LIN {X 0,Y 383.71,Z 437.211,A -85,B 0,C 180,E1 -14302.123,E2 -14302.123} C_VEL
LIN {X 0,Y 386.289,Z 439.249,A -85,B 0,C 180,E1 -14303.895,E2 -14303.895} C_VEL
LIN {X 0,Y 388.386,Z 440.41,A -85,B 0,C 180,E1 -14305.849,E2 -14305.849} C_VEL
LIN {X 0,Y 389.529,Z 440.796,A -85,B 0,C 180,E1 -14307.433,E2 -14307.433} C_VEL
LIN {X 0,Y 390.099,Z 441.222,A -85,B 0,C 180,E1 -14308.967,E2 -14308.967} C_VEL
LIN {X 0,Y 390.27,Z 441.152,A -85,B 0,C 180,E1 -14310,E2 -14310} C_VEL
LIN {X 0,Y 389.995,Z 441.089,A -85,B 0,C 180,E1 -14311.549,E2 -14311.549} C_VEL
LIN {X 0,Y 389.238,Z 440.657,A -85,B 0,C 180,E1 -14313.105,E2 -14313.105} C_VEL
LIN {X 0,Y 387.614,Z 440.065,A -85,B 0,C 180,E1 -14314.94,E2 -14314.94} C_VEL
LIN {X 0,Y 385.471,Z 438.704,A -85,B 0,C 180,E1 -14316.685,E2 -14316.685} C_VEL
LIN {X 0,Y 383.224,Z 436.724,A -85,B 0,C 180,E1 -14318.162,E2 -14318.162} C_VEL
LIN {X 0,Y 380.545,Z 433.68,A -85,B 0,C 180,E1 -14319.669,E2 -14319.669} C_VEL
LIN {X 0,Y 377.343,Z 431.776,A -85,B 0,C 180,E1 -14321.118,E2 -14321.118} C_VEL
LIN {X 0,Y 373.996,Z 428.62,A -85,B 0,C 180,E1 -14322.503,E2 -14322.503} C_VEL
LIN {X 0,Y 371.832,Z 426.329,A -85,B 0,C 180,E1 -14323.336,E2 -14323.336} C_VEL
LIN {X 0,Y 368.143,Z 423.337,A -85,B 0,C 180,E1 -14324.583,E2 -14324.583} C_VEL
LIN {X 0,Y 365.094,Z 419.876,A -85,B 0,C 180,E1 -14325.58,E2 -14325.58} C_VEL
LIN {X 0,Y 361.446,Z 416.759,A -85,B 0,C 180,E1 -14326.666,E2 -14326.666} C_VEL
LIN {X 0,Y 358.551,Z 413.451,A -85,B 0,C 180,E1 -14327.482,E2 -14327.482} C_VEL
LIN {X 0,Y 355.376,Z 410.462,A -85,B 0,C 180,E1 -14328.333,E2 -14328.333} C_VEL
LIN {X 0,Y 353.051,Z 407.518,A -85,B 0,C 180,E1 -14328.94,E2 -14328.94} C_VEL
LIN {X 0,Y 350.002,Z 404.381,A -85,B 0,C 180,E1 -14329.706,E2 -14329.706} C_VEL
LIN {X 0,Y 348.216,Z 401.952,A -85,B 0,C 180,E1 -14330.137,E2 -14330.137} C_VEL
LIN {X 0,Y 345.497,Z 399.057,A -85,B 0,C 180,E1 -14330.784,E2 -14330.784} C_VEL
LIN {X 0,Y 344.016,Z 396.656,A -85,B 0,C 180,E1 -14331.146,E2 -14331.146} C_VEL
LIN {X 0,Y 341.851,Z 394.52,A -85,B 0,C 180,E1 -14331.605,E2 -14331.605} C_VEL
LIN {X 0,Y 340.819,Z 392.08,A -85,B 0,C 180,E1 -14331.984,E2 -14331.984} C_VEL
LIN {X 0,Y 340.741,Z 391.556,A -85,B 0,C 180,E1 -14332.43,E2 -14332.43} C_VEL
LIN {X 0,Y 340.768,Z 391.54,A -85,B 0,C 180,E1 -14335.664,E2 -14335.664} C_VEL
LIN {X 0,Y 340.737,Z 391.527,A -85,B 0,C 180,E1 -14338.319,E2 -14338.319} C_VEL
LIN {X 0,Y 340.698,Z 391.542,A -85,B 0,C 180,E1 -14341.044,E2 -14341.044} C_VEL
LIN {X 0,Y 340.713,Z 391.518,A -85,B 0,C 180,E1 -14345.279,E2 -14345.279} C_VEL
LIN {X 0,Y 340.72,Z 391.546,A -85,B 0,C 180,E1 -14348.389,E2 -14348.389} C_VEL
LIN {X 0,Y 340.699,Z 391.499,A -85,B 0,C 180,E1 -14352.047,E2 -14352.047} C_VEL
LIN {X 0,Y 340.688,Z 391.544,A -85,B 0,C 180,E1 -14355.463,E2 -14355.463} C_VEL
LIN {X 0,Y 340.697,Z 391.534,A -85,B 0,C 180,E1 -14358.693,E2 -14358.693} C_VEL
LIN {X 0,Y 340.734,Z 391.541,A -85,B 0,C 180,E1 -14361.774,E2 -14361.774} C_VEL
LIN {X 0,Y 340.716,Z 391.524,A -85,B 0,C 180,E1 -14365.596,E2 -14365.596} C_VEL
LIN {X 0,Y 340.717,Z 391.542,A -85,B 0,C 180,E1 -14369.566,E2 -14369.566} C_VEL
LIN {X 0,Y 340.799,Z 391.513,A -85,B 0,C 180,E1 -14373.02,E2 -14373.02} C_VEL
LIN {X 0,Y 340.755,Z 391.53,A -85,B 0,C 180,E1 -14374.691,E2 -14374.691} C_VEL
LIN {X 0,Y 340.072,Z 391.623,A -85,B 0,C 180,E1 -14375.678,E2 -14375.678} C_VEL
LIN {X 0,Y 337.177,Z 391.982,A -85,B 0,C 180,E1 -14377.283,E2 -14377.283} C_VEL
LIN {X 0,Y 334.755,Z 392.275,A -85,B 0,C 180,E1 -14378.582,E2 -14378.582} C_VEL
LIN {X 0,Y 333.756,Z 392.392,A -85,B 0,C 180,E1 -14379.589,E2 -14379.589} C_VEL
LIN {X 0,Y 333.695,Z 392.393,A -85,B 0,C 180,E1 -14379.93,E2 -14379.93} C_VEL
LIN {X 0,Y 333.74,Z 392.401,A -85,B 0,C 180,E1 -14382.854,E2 -14382.854} C_VEL
LIN {X 0,Y 333.792,Z 392.401,A -85,B 0,C 180,E1 -14386.609,E2 -14386.609} C_VEL
LIN {X 0,Y 333.858,Z 392.366,A -85,B 0,C 180,E1 -14390.306,E2 -14390.306} C_VEL
LIN {X 0,Y 334.019,Z 392.371,A -85,B 0,C 180,E1 -14392.748,E2 -14392.748} C_VEL
LIN {X 0,Y 333.807,Z 392.402,A -85,B 0,C 180,E1 -14395.17,E2 -14395.17} C_VEL
LIN {X 0,Y 334.102,Z 392.353,A -85,B 0,C 180,E1 -14397.589,E2 -14397.589} C_VEL
LIN {X 0,Y 334.223,Z 392.318,A -85,B 0,C 180,E1 -14400.001,E2 -14400.001} C_VEL
LIN {X 0,Y 334.102,Z 392.358,A -85,B 0,C 180,E1 -14402.412,E2 -14402.412} C_VEL
LIN {X 0,Y 334.022,Z 392.364,A -85,B 0,C 180,E1 -14407.253,E2 -14407.253} C_VEL
LIN {X 0,Y 333.829,Z 392.38,A -85,B 0,C 180,E1 -14410.923,E2 -14410.923} C_VEL
LIN {X 0,Y 333.804,Z 392.401,A -85,B 0,C 180,E1 -14414.635,E2 -14414.635} C_VEL
LIN {X 0,Y 333.792,Z 392.376,A -85,B 0,C 180,E1 -14418.656,E2 -14418.656} C_VEL
LIN {X 0,Y 333.689,Z 392.419,A -85,B 0,C 180,E1 -14422.279,E2 -14422.279} C_VEL
LIN {X 0,Y 333.733,Z 392.389,A -85,B 0,C 180,E1 -14426.247,E2 -14426.247} C_VEL
LIN {X 0,Y 333.709,Z 392.412,A -85,B 0,C 180,E1 -14428.973,E2 -14428.973} C_VEL
LIN {X 0,Y 333.649,Z 392.412,A -85,B 0,C 180,E1 -14432.59,E2 -14432.59} C_VEL
LIN {X 0,Y 333.675,Z 392.417,A -85,B 0,C 180,E1 -14436.14,E2 -14436.14} C_VEL
LIN {X 0,Y 333.683,Z 392.411,A -85,B 0,C 180,E1 -14439.188,E2 -14439.188} C_VEL
LIN {X 0,Y 333.701,Z 392.417,A -85,B 0,C 180,E1 -14442.514,E2 -14442.514} C_VEL
LIN {X 0,Y 333.634,Z 392.428,A -85,B 0,C 180,E1 -14445.962,E2 -14445.962} C_VEL
LIN {X 0,Y 333.646,Z 392.399,A -85,B 0,C 180,E1 -14449.316,E2 -14449.316} C_VEL
LIN {X 0,Y 333.666,Z 392.412,A -85,B 0,C 180,E1 -14453.169,E2 -14453.169} C_VEL
LIN {X 0,Y 333.704,Z 392.564,A -85,B 0,C 180,E1 -14456.865,E2 -14456.865} C_VEL
LIN {X 0,Y 335.043,Z 398.947,A -85,B 0,C 180,E1 -14459.321,E2 -14459.321} C_VEL
LIN {X 0,Y 336.889,Z 408.593,A -85,B 0,C 180,E1 -14462.681,E2 -14462.681} C_VEL
LIN {X 0,Y 337.083,Z 412.536,A -85,B 0,C 180,E1 -14464.035,E2 -14464.035} C_VEL
LIN {X 0,Y 336.305,Z 418.399,A -85,B 0,C 180,E1 -14465.916,E2 -14465.916} C_VEL
LIN {X 0,Y 337.098,Z 422.527,A -85,B 0,C 180,E1 -14466.137,E2 -14466.137} C_VEL
LIN {X 0,Y 341.775,Z 445.874,A -85,B 0,C 180,E1 -14467.003,E2 -14467.003} C_VEL
LIN {X 0,Y 343.729,Z 457.616,A -85,B 0,C 180,E1 -14467.4,E2 -14467.4} C_VEL
LIN {X 0,Y 342.424,Z 523.377,A -85,B 0,C 180,E1 -14468.794,E2 -14468.794} C_VEL
LIN {X 0,Y 341.954,Z 533.264,A -85,B 0,C 180,E1 -14469.118,E2 -14469.118} C_VEL
LIN {X 0,Y 341.257,Z 543.248,A -85,B 0,C 180,E1 -14469.586,E2 -14469.586} C_VEL
LIN {X 0,Y 340.344,Z 553.602,A -85,B 0,C 180,E1 -14470.237,E2 -14470.237} C_VEL
LIN {X 0,Y 339.437,Z 562.747,A -85,B 0,C 180,E1 -14470.968,E2 -14470.968} C_VEL
LIN {X 0,Y 338.37,Z 571.746,A -85,B 0,C 180,E1 -14471.848,E2 -14471.848} C_VEL
LIN {X 0,Y 337.296,Z 580.473,A -85,B 0,C 180,E1 -14472.884,E2 -14472.884} C_VEL
LIN {X 0,Y 336.298,Z 588.415,A -85,B 0,C 180,E1 -14474.013,E2 -14474.013} C_VEL
LIN {X 0,Y 335.243,Z 596.692,A -85,B 0,C 180,E1 -14475.43,E2 -14475.43} C_VEL
LIN {X 0,Y 334.488,Z 602.684,A -85,B 0,C 180,E1 -14476.637,E2 -14476.637} C_VEL
LIN {X 0,Y 333.587,Z 608.993,A -85,B 0,C 180,E1 -14478.147,E2 -14478.147} C_VEL
LIN {X 0,Y 333.006,Z 614.269,A -85,B 0,C 180,E1 -14479.666,E2 -14479.666} C_VEL
LIN {X 0,Y 332.464,Z 619.364,A -85,B 0,C 180,E1 -14481.491,E2 -14481.491} C_VEL
LIN {X 0,Y 332.121,Z 623.328,A -85,B 0,C 180,E1 -14483.317,E2 -14483.317} C_VEL
LIN {X 0,Y 331.981,Z 626.264,A -85,B 0,C 180,E1 -14485.143,E2 -14485.143} C_VEL
LIN {X 0,Y 331.97,Z 627.765,A -85,B 0,C 180,E1 -14486.359,E2 -14486.359} C_VEL
LIN {X 0,Y 331.913,Z 629.287,A -85,B 0,C 180,E1 -14488.787,E2 -14488.787} C_VEL
LIN {X 0,Y 331.953,Z 629.567,A -85,B 0,C 180,E1 -14490,E2 -14490} C_VEL
LIN {X 0,Y 331.916,Z 628.691,A -85,B 0,C 180,E1 -14492.427,E2 -14492.427} C_VEL
LIN {X 0,Y 331.97,Z 627.764,A -85,B 0,C 180,E1 -14493.642,E2 -14493.642} C_VEL
LIN {X 0,Y 332.039,Z 624.416,A -85,B 0,C 180,E1 -14496.075,E2 -14496.075} C_VEL
LIN {X 0,Y 332.335,Z 620.79,A -85,B 0,C 180,E1 -14497.901,E2 -14497.901} C_VEL
LIN {X 0,Y 332.793,Z 616.057,A -85,B 0,C 180,E1 -14499.727,E2 -14499.727} C_VEL
LIN {X 0,Y 333.442,Z 610.083,A -85,B 0,C 180,E1 -14501.551,E2 -14501.551} C_VEL
LIN {X 0,Y 334.289,Z 603.992,A -85,B 0,C 180,E1 -14503.062,E2 -14503.062} C_VEL
LIN {X 0,Y 335.081,Z 598.251,A -85,B 0,C 180,E1 -14504.267,E2 -14504.267} C_VEL
LIN {X 0,Y 336.001,Z 591.595,A -85,B 0,C 180,E1 -14505.467,E2 -14505.467} C_VEL
LIN {X 0,Y 336.919,Z 583.763,A -85,B 0,C 180,E1 -14506.668,E2 -14506.668} C_VEL
LIN {X 0,Y 337.935,Z 575.68,A -85,B 0,C 180,E1 -14507.707,E2 -14507.707} C_VEL
LIN {X 0,Y 339.078,Z 565.919,A -85,B 0,C 180,E1 -14508.74,E2 -14508.74} C_VEL
LIN {X 0,Y 339.985,Z 557.529,A -85,B 0,C 180,E1 -14509.471,E2 -14509.471} C_VEL
LIN {X 0,Y 340.903,Z 547.022,A -85,B 0,C 180,E1 -14510.201,E2 -14510.201} C_VEL
LIN {X 0,Y 341.734,Z 536.691,A -85,B 0,C 180,E1 -14510.739,E2 -14510.739} C_VEL
LIN {X 0,Y 342.353,Z 525.97,A -85,B 0,C 180,E1 -14511.133,E2 -14511.133} C_VEL
LIN {X 0,Y 342.826,Z 503.188,A -85,B 0,C 180,E1 -14511.654,E2 -14511.654} C_VEL
LIN {X 0,Y 343.607,Z 456.424,A -85,B 0,C 180,E1 -14512.635,E2 -14512.635} C_VEL
LIN {X 0,Y 339.119,Z 431.992,A -85,B 0,C 180,E1 -14513.499,E2 -14513.499} C_VEL
LIN {X 0,Y 336.289,Z 418.735,A -85,B 0,C 180,E1 -14514.04,E2 -14514.04} C_VEL
LIN {X 0,Y 336.392,Z 417.243,A -85,B 0,C 180,E1 -14514.403,E2 -14514.403} C_VEL
LIN {X 0,Y 337.206,Z 411.413,A -85,B 0,C 180,E1 -14516.336,E2 -14516.336} C_VEL
LIN {X 0,Y 336.18,Z 404.578,A -85,B 0,C 180,E1 -14518.739,E2 -14518.739} C_VEL
LIN {X 0,Y 334.245,Z 395.104,A -85,B 0,C 180,E1 -14522.173,E2 -14522.173} C_VEL
LIN {X 0,Y 333.705,Z 392.506,A -85,B 0,C 180,E1 -14523.201,E2 -14523.201} C_VEL
LIN {X 0,Y 333.668,Z 392.412,A -85,B 0,C 180,E1 -14526.832,E2 -14526.832} C_VEL
LIN {X 0,Y 333.648,Z 392.398,A -85,B 0,C 180,E1 -14530.767,E2 -14530.767} C_VEL
LIN {X 0,Y 333.645,Z 392.424,A -85,B 0,C 180,E1 -14534.259,E2 -14534.259} C_VEL
LIN {X 0,Y 333.707,Z 392.417,A -85,B 0,C 180,E1 -14537.628,E2 -14537.628} C_VEL
LIN {X 0,Y 333.685,Z 392.412,A -85,B 0,C 180,E1 -14541.195,E2 -14541.195} C_VEL
LIN {X 0,Y 333.687,Z 392.405,A -85,B 0,C 180,E1 -14545.225,E2 -14545.225} C_VEL
LIN {X 0,Y 333.645,Z 392.422,A -85,B 0,C 180,E1 -14548.223,E2 -14548.223} C_VEL
LIN {X 0,Y 333.713,Z 392.411,A -85,B 0,C 180,E1 -14551.027,E2 -14551.027} C_VEL
LIN {X 0,Y 333.736,Z 392.389,A -85,B 0,C 180,E1 -14553.753,E2 -14553.753} C_VEL
LIN {X 0,Y 333.72,Z 392.412,A -85,B 0,C 180,E1 -14557.913,E2 -14557.913} C_VEL
LIN {X 0,Y 333.793,Z 392.376,A -85,B 0,C 180,E1 -14561.589,E2 -14561.589} C_VEL
LIN {X 0,Y 333.808,Z 392.402,A -85,B 0,C 180,E1 -14565.576,E2 -14565.576} C_VEL
LIN {X 0,Y 333.833,Z 392.379,A -85,B 0,C 180,E1 -14569.077,E2 -14569.077} C_VEL
LIN {X 0,Y 334.026,Z 392.364,A -85,B 0,C 180,E1 -14572.747,E2 -14572.747} C_VEL
LIN {X 0,Y 333.81,Z 392.403,A -85,B 0,C 180,E1 -14575.168,E2 -14575.168} C_VEL
LIN {X 0,Y 334.106,Z 392.357,A -85,B 0,C 180,E1 -14577.588,E2 -14577.588} C_VEL
LIN {X 0,Y 334.225,Z 392.317,A -85,B 0,C 180,E1 -14579.999,E2 -14579.999} C_VEL
LIN {X 0,Y 334.106,Z 392.353,A -85,B 0,C 180,E1 -14582.41,E2 -14582.41} C_VEL
LIN {X 0,Y 334.023,Z 392.37,A -85,B 0,C 180,E1 -14587.252,E2 -14587.252} C_VEL
LIN {X 0,Y 333.834,Z 392.372,A -85,B 0,C 180,E1 -14590.921,E2 -14590.921} C_VEL
LIN {X 0,Y 333.806,Z 392.403,A -85,B 0,C 180,E1 -14594.634,E2 -14594.634} C_VEL
LIN {X 0,Y 333.793,Z 392.38,A -85,B 0,C 180,E1 -14598.654,E2 -14598.654} C_VEL
LIN {X 0,Y 333.69,Z 392.416,A -85,B 0,C 180,E1 -14602.278,E2 -14602.278} C_VEL
LIN {X 0,Y 333.732,Z 392.398,A -85,B 0,C 180,E1 -14606.246,E2 -14606.246} C_VEL
LIN {X 0,Y 333.687,Z 392.407,A -85,B 0,C 180,E1 -14608.974,E2 -14608.974} C_VEL
LIN {X 0,Y 333.64,Z 392.422,A -85,B 0,C 180,E1 -14612.586,E2 -14612.586} C_VEL
LIN {X 0,Y 333.674,Z 392.416,A -85,B 0,C 180,E1 -14616.138,E2 -14616.138} C_VEL
LIN {X 0,Y 333.644,Z 392.42,A -85,B 0,C 180,E1 -14619.192,E2 -14619.192} C_VEL
LIN {X 0,Y 333.63,Z 392.423,A -85,B 0,C 180,E1 -14622.5,E2 -14622.5} C_VEL
LIN {X 0,Y 333.617,Z 392.406,A -85,B 0,C 180,E1 -14625.959,E2 -14625.959} C_VEL
LIN {X 0,Y 333.651,Z 392.388,A -85,B 0,C 180,E1 -14629.313,E2 -14629.313} C_VEL
LIN {X 0,Y 333.657,Z 392.424,A -85,B 0,C 180,E1 -14632.35,E2 -14632.35} C_VEL
LIN {X 0,Y 333.671,Z 392.392,A -85,B 0,C 180,E1 -14635.341,E2 -14635.341} C_VEL
LIN {X 0,Y 333.699,Z 392.403,A -85,B 0,C 180,E1 -14639.71,E2 -14639.71} C_VEL
LIN {X 0,Y 333.741,Z 392.41,A -85,B 0,C 180,E1 -14642.401,E2 -14642.401} C_VEL
LIN {X 0,Y 333.723,Z 392.417,A -85,B 0,C 180,E1 -14645.09,E2 -14645.09} C_VEL
LIN {X 0,Y 333.715,Z 392.563,A -85,B 0,C 180,E1 -14646.635,E2 -14646.635} C_VEL
LIN {X 0,Y 333.903,Z 393.474,A -85,B 0,C 180,E1 -14646.906,E2 -14646.906} C_VEL
LIN {X 0,Y 335.441,Z 396.247,A -85,B 0,C 180,E1 -14647.293,E2 -14647.293} C_VEL
LIN {X 0,Y 337.241,Z 398.134,A -85,B 0,C 180,E1 -14647.649,E2 -14647.649} C_VEL
LIN {X 0,Y 339.605,Z 401.544,A -85,B 0,C 180,E1 -14648.193,E2 -14648.193} C_VEL
LIN {X 0,Y 341.244,Z 403.295,A -85,B 0,C 180,E1 -14648.55,E2 -14648.55} C_VEL
LIN {X 0,Y 344.183,Z 407.005,A -85,B 0,C 180,E1 -14649.205,E2 -14649.205} C_VEL
LIN {X 0,Y 346.049,Z 408.972,A -85,B 0,C 180,E1 -14649.649,E2 -14649.649} C_VEL
LIN {X 0,Y 349.255,Z 412.734,A -85,B 0,C 180,E1 -14650.409,E2 -14650.409} C_VEL
LIN {X 0,Y 351.179,Z 414.637,A -85,B 0,C 180,E1 -14650.881,E2 -14650.881} C_VEL
LIN {X 0,Y 354.984,Z 418.848,A -85,B 0,C 180,E1 -14651.859,E2 -14651.859} C_VEL
LIN {X 0,Y 357.006,Z 420.704,A -85,B 0,C 180,E1 -14652.398,E2 -14652.398} C_VEL
LIN {X 0,Y 361.089,Z 424.937,A -85,B 0,C 180,E1 -14653.544,E2 -14653.544} C_VEL
LIN {X 0,Y 363.83,Z 427.288,A -85,B 0,C 180,E1 -14654.364,E2 -14654.364} C_VEL
LIN {X 0,Y 367.521,Z 431.12,A -85,B 0,C 180,E1 -14655.552,E2 -14655.552} C_VEL
LIN {X 0,Y 371.229,Z 434.051,A -85,B 0,C 180,E1 -14656.812,E2 -14656.812} C_VEL
LIN {X 0,Y 374.886,Z 437.757,A -85,B 0,C 180,E1 -14658.241,E2 -14658.241} C_VEL
LIN {X 0,Y 378.477,Z 440.221,A -85,B 0,C 180,E1 -14659.786,E2 -14659.786} C_VEL
LIN {X 0,Y 379.779,Z 441.047,A -85,B 0,C 180,E1 -14660.413,E2 -14660.413} C_VEL
LIN {X 0,Y 382.384,Z 443.977,A -85,B 0,C 180,E1 -14661.88,E2 -14661.88} C_VEL
LIN {X 0,Y 384.714,Z 445.9,A -85,B 0,C 180,E1 -14663.407,E2 -14663.407} C_VEL
LIN {X 0,Y 387.037,Z 447.233,A -85,B 0,C 180,E1 -14665.318,E2 -14665.318} C_VEL
LIN {X 0,Y 388.664,Z 447.822,A -85,B 0,C 180,E1 -14667.428,E2 -14667.428} C_VEL
LIN {X 0,Y 389.239,Z 448.261,A -85,B 0,C 180,E1 -14668.965,E2 -14668.965} C_VEL
LIN {X 0,Y 389.407,Z 448.18,A -85,B 0,C 180,E1 -14670,E2 -14670} C_VEL
LIN {X 0,Y 389.126,Z 448.137,A -85,B 0,C 180,E1 -14671.552,E2 -14671.552} C_VEL
LIN {X 0,Y 388.36,Z 447.704,A -85,B 0,C 180,E1 -14673.112,E2 -14673.112} C_VEL
LIN {X 0,Y 386.735,Z 447.105,A -85,B 0,C 180,E1 -14674.942,E2 -14674.942} C_VEL
LIN {X 0,Y 384.555,Z 445.811,A -85,B 0,C 180,E1 -14676.701,E2 -14676.701} C_VEL
LIN {X 0,Y 382.058,Z 443.694,A -85,B 0,C 180,E1 -14678.309,E2 -14678.309} C_VEL
LIN {X 0,Y 379.211,Z 440.56,A -85,B 0,C 180,E1 -14679.866,E2 -14679.866} C_VEL
LIN {X 0,Y 375.944,Z 438.624,A -85,B 0,C 180,E1 -14681.307,E2 -14681.307} C_VEL
LIN {X 0,Y 372.543,Z 435.544,A -85,B 0,C 180,E1 -14682.676,E2 -14682.676} C_VEL
LIN {X 0,Y 370.203,Z 433.07,A -85,B 0,C 180,E1 -14683.569,E2 -14683.569} C_VEL
LIN {X 0,Y 366.134,Z 429.818,A -85,B 0,C 180,E1 -14684.914,E2 -14684.914} C_VEL
LIN {X 0,Y 362.656,Z 426.153,A -85,B 0,C 180,E1 -14685.994,E2 -14685.994} C_VEL
LIN {X 0,Y 358.914,Z 422.914,A -85,B 0,C 180,E1 -14687.059,E2 -14687.059} C_VEL
LIN {X 0,Y 355.812,Z 419.521,A -85,B 0,C 180,E1 -14687.928,E2 -14687.928} C_VEL
LIN {X 0,Y 352.062,Z 415.824,A -85,B 0,C 180,E1 -14688.881,E2 -14688.881} C_VEL
LIN {X 0,Y 350.012,Z 413.398,A -85,B 0,C 180,E1 -14689.415,E2 -14689.415} C_VEL
LIN {X 0,Y 346.537,Z 409.698,A -85,B 0,C 180,E1 -14690.229,E2 -14690.229} C_VEL
LIN {X 0,Y 344.964,Z 407.748,A -85,B 0,C 180,E1 -14690.613,E2 -14690.613} C_VEL
LIN {X 0,Y 341.952,Z 404.421,A -85,B 0,C 180,E1 -14691.286,E2 -14691.286} C_VEL
LIN {X 0,Y 340.285,Z 402.167,A -85,B 0,C 180,E1 -14691.661,E2 -14691.661} C_VEL
LIN {X 0,Y 337.899,Z 399.318,A -85,B 0,C 180,E1 -14692.197,E2 -14692.197} C_VEL
LIN {X 0,Y 336.544,Z 397.283,A -85,B 0,C 180,E1 -14692.493,E2 -14692.493} C_VEL
LIN {X 0,Y 334.615,Z 395.151,A -85,B 0,C 180,E1 -14692.878,E2 -14692.878} C_VEL
LIN {X 0,Y 333.8,Z 393.074,A -85,B 0,C 180,E1 -14693.17,E2 -14693.17} C_VEL
LIN {X 0,Y 333.679,Z 392.494,A -85,B 0,C 180,E1 -14693.424,E2 -14693.424} C_VEL
LIN {X 0,Y 333.731,Z 392.416,A -85,B 0,C 180,E1 -14696.246,E2 -14696.246} C_VEL
LIN {X 0,Y 333.706,Z 392.397,A -85,B 0,C 180,E1 -14698.972,E2 -14698.972} C_VEL
LIN {X 0,Y 333.637,Z 392.419,A -85,B 0,C 180,E1 -14702.587,E2 -14702.587} C_VEL
LIN {X 0,Y 333.672,Z 392.406,A -85,B 0,C 180,E1 -14706.138,E2 -14706.138} C_VEL
LIN {X 0,Y 333.668,Z 392.415,A -85,B 0,C 180,E1 -14709.188,E2 -14709.188} C_VEL
LIN {X 0,Y 333.631,Z 392.38,A -85,B 0,C 180,E1 -14712.501,E2 -14712.501} C_VEL
LIN {X 0,Y 333.637,Z 392.423,A -85,B 0,C 180,E1 -14715.963,E2 -14715.963} C_VEL
LIN {X 0,Y 333.649,Z 392.409,A -85,B 0,C 180,E1 -14719.314,E2 -14719.314} C_VEL
LIN {X 0,Y 333.651,Z 392.426,A -85,B 0,C 180,E1 -14722.35,E2 -14722.35} C_VEL
LIN {X 0,Y 333.667,Z 392.402,A -85,B 0,C 180,E1 -14725.341,E2 -14725.341} C_VEL
LIN {X 0,Y 333.696,Z 392.417,A -85,B 0,C 180,E1 -14729.71,E2 -14729.71} C_VEL
LIN {X 0,Y 333.738,Z 392.39,A -85,B 0,C 180,E1 -14732.402,E2 -14732.402} C_VEL
LIN {X 0,Y 333.72,Z 392.413,A -85,B 0,C 180,E1 -14735.091,E2 -14735.091} C_VEL
LIN {X 0,Y 333.673,Z 392.406,A -85,B 0,C 180,E1 -14739.02,E2 -14739.02} C_VEL
LIN {X 0,Y 333.695,Z 392.393,A -85,B 0,C 180,E1 -14739.93,E2 -14739.93} C_VEL
LIN {X 0,Y 333.086,Z 392.468,A -85,B 0,C 180,E1 -14740.937,E2 -14740.937} C_VEL
LIN {X 0,Y 330.262,Z 392.831,A -85,B 0,C 180,E1 -14742.576,E2 -14742.576} C_VEL
LIN {X 0,Y 327.847,Z 393.142,A -85,B 0,C 180,E1 -14743.904,E2 -14743.904} C_VEL
LIN {X 0,Y 326.825,Z 393.274,A -85,B 0,C 180,E1 -14744.932,E2 -14744.932} C_VEL
LIN {X 0,Y 326.752,Z 393.282,A -85,B 0,C 180,E1 -14745.28,E2 -14745.28} C_VEL
LIN {X 0,Y 326.766,Z 393.254,A -85,B 0,C 180,E1 -14748.84,E2 -14748.84} C_VEL
LIN {X 0,Y 326.973,Z 393.245,A -85,B 0,C 180,E1 -14752.591,E2 -14752.591} C_VEL
LIN {X 0,Y 326.774,Z 393.278,A -85,B 0,C 180,E1 -14755.066,E2 -14755.066} C_VEL
LIN {X 0,Y 327.043,Z 393.232,A -85,B 0,C 180,E1 -14757.537,E2 -14757.537} C_VEL
LIN {X 0,Y 327.175,Z 393.195,A -85,B 0,C 180,E1 -14760.001,E2 -14760.001} C_VEL
LIN {X 0,Y 327.043,Z 393.237,A -85,B 0,C 180,E1 -14762.464,E2 -14762.464} C_VEL
LIN {X 0,Y 326.992,Z 393.248,A -85,B 0,C 180,E1 -14766.17,E2 -14766.17} C_VEL
LIN {X 0,Y 326.91,Z 393.229,A -85,B 0,C 180,E1 -14768.656,E2 -14768.656} C_VEL
LIN {X 0,Y 326.73,Z 393.278,A -85,B 0,C 180,E1 -14772.422,E2 -14772.422} C_VEL
LIN {X 0,Y 326.75,Z 393.277,A -85,B 0,C 180,E1 -14774.958,E2 -14774.958} C_VEL
LIN {X 0,Y 326.729,Z 393.255,A -85,B 0,C 180,E1 -14778.839,E2 -14778.839} C_VEL
LIN {X 0,Y 326.617,Z 393.297,A -85,B 0,C 180,E1 -14782.788,E2 -14782.788} C_VEL
LIN {X 0,Y 326.687,Z 393.274,A -85,B 0,C 180,E1 -14785.485,E2 -14785.485} C_VEL
LIN {X 0,Y 326.659,Z 393.291,A -85,B 0,C 180,E1 -14789.66,E2 -14789.66} C_VEL
LIN {X 0,Y 326.62,Z 393.286,A -85,B 0,C 180,E1 -14792.949,E2 -14792.949} C_VEL
LIN {X 0,Y 326.632,Z 393.297,A -85,B 0,C 180,E1 -14797.047,E2 -14797.047} C_VEL
LIN {X 0,Y 326.634,Z 393.287,A -85,B 0,C 180,E1 -14800.203,E2 -14800.203} C_VEL
LIN {X 0,Y 326.64,Z 393.293,A -85,B 0,C 180,E1 -14803.513,E2 -14803.513} C_VEL
LIN {X 0,Y 326.585,Z 393.303,A -85,B 0,C 180,E1 -14807.027,E2 -14807.027} C_VEL
LIN {X 0,Y 326.611,Z 393.288,A -85,B 0,C 180,E1 -14810.774,E2 -14810.774} C_VEL
LIN {X 0,Y 326.613,Z 393.286,A -85,B 0,C 180,E1 -14814.481,E2 -14814.481} C_VEL
LIN {X 0,Y 326.68,Z 393.53,A -85,B 0,C 180,E1 -14816.488,E2 -14816.488} C_VEL
LIN {X 0,Y 328.294,Z 401.164,A -85,B 0,C 180,E1 -14819.441,E2 -14819.441} C_VEL
LIN {X 0,Y 329.992,Z 410.363,A -85,B 0,C 180,E1 -14822.75,E2 -14822.75} C_VEL
LIN {X 0,Y 330.23,Z 412.337,A -85,B 0,C 180,E1 -14823.454,E2 -14823.454} C_VEL
LIN {X 0,Y 329.461,Z 418.216,A -85,B 0,C 180,E1 -14825.387,E2 -14825.387} C_VEL
LIN {X 0,Y 330.324,Z 422.406,A -85,B 0,C 180,E1 -14825.618,E2 -14825.618} C_VEL
LIN {X 0,Y 335.301,Z 447.238,A -85,B 0,C 180,E1 -14826.568,E2 -14826.568} C_VEL
LIN {X 0,Y 337.175,Z 458.618,A -85,B 0,C 180,E1 -14826.962,E2 -14826.962} C_VEL
LIN {X 0,Y 335.831,Z 523.19,A -85,B 0,C 180,E1 -14828.356,E2 -14828.356} C_VEL
LIN {X 0,Y 335.343,Z 533.069,A -85,B 0,C 180,E1 -14828.686,E2 -14828.686} C_VEL
LIN {X 0,Y 334.613,Z 543.053,A -85,B 0,C 180,E1 -14829.162,E2 -14829.162} C_VEL
LIN {X 0,Y 333.656,Z 553.406,A -85,B 0,C 180,E1 -14829.824,E2 -14829.824} C_VEL
LIN {X 0,Y 332.716,Z 562.551,A -85,B 0,C 180,E1 -14830.569,E2 -14830.569} C_VEL
LIN {X 0,Y 331.624,Z 571.551,A -85,B 0,C 180,E1 -14831.465,E2 -14831.465} C_VEL
LIN {X 0,Y 330.503,Z 580.277,A -85,B 0,C 180,E1 -14832.521,E2 -14832.521} C_VEL
LIN {X 0,Y 329.348,Z 588.969,A -85,B 0,C 180,E1 -14833.795,E2 -14833.795} C_VEL
LIN {X 0,Y 328.343,Z 596.496,A -85,B 0,C 180,E1 -14835.117,E2 -14835.117} C_VEL
LIN {X 0,Y 327.569,Z 602.489,A -85,B 0,C 180,E1 -14836.35,E2 -14836.35} C_VEL
LIN {X 0,Y 326.618,Z 608.798,A -85,B 0,C 180,E1 -14837.89,E2 -14837.89} C_VEL
LIN {X 0,Y 325.98,Z 614.073,A -85,B 0,C 180,E1 -14839.441,E2 -14839.441} C_VEL
LIN {X 0,Y 325.405,Z 619.167,A -85,B 0,C 180,E1 -14841.305,E2 -14841.305} C_VEL
LIN {X 0,Y 325.056,Z 623.133,A -85,B 0,C 180,E1 -14843.171,E2 -14843.171} C_VEL
LIN {X 0,Y 324.895,Z 626.068,A -85,B 0,C 180,E1 -14845.037,E2 -14845.037} C_VEL
LIN {X 0,Y 324.877,Z 627.57,A -85,B 0,C 180,E1 -14846.279,E2 -14846.279} C_VEL
LIN {X 0,Y 324.822,Z 629.092,A -85,B 0,C 180,E1 -14848.761,E2 -14848.761} C_VEL
LIN {X 0,Y 324.859,Z 629.372,A -85,B 0,C 180,E1 -14850,E2 -14850} C_VEL
LIN {X 0,Y 324.836,Z 628.497,A -85,B 0,C 180,E1 -14852.48,E2 -14852.48} C_VEL
LIN {X 0,Y 324.876,Z 627.569,A -85,B 0,C 180,E1 -14853.721,E2 -14853.721} C_VEL
LIN {X 0,Y 324.96,Z 624.22,A -85,B 0,C 180,E1 -14856.208,E2 -14856.208} C_VEL
LIN {X 0,Y 325.266,Z 620.594,A -85,B 0,C 180,E1 -14858.074,E2 -14858.074} C_VEL
LIN {X 0,Y 325.78,Z 615.862,A -85,B 0,C 180,E1 -14859.938,E2 -14859.938} C_VEL
LIN {X 0,Y 326.456,Z 609.887,A -85,B 0,C 180,E1 -14861.801,E2 -14861.801} C_VEL
LIN {X 0,Y 327.338,Z 603.796,A -85,B 0,C 180,E1 -14863.345,E2 -14863.345} C_VEL
LIN {X 0,Y 328.167,Z 598.055,A -85,B 0,C 180,E1 -14864.575,E2 -14864.575} C_VEL
LIN {X 0,Y 329.142,Z 591.399,A -85,B 0,C 180,E1 -14865.798,E2 -14865.798} C_VEL
LIN {X 0,Y 330.062,Z 583.788,A -85,B 0,C 180,E1 -14866.993,E2 -14866.993} C_VEL
LIN {X 0,Y 331.151,Z 575.484,A -85,B 0,C 180,E1 -14868.083,E2 -14868.083} C_VEL
LIN {X 0,Y 332.349,Z 565.723,A -85,B 0,C 180,E1 -14869.134,E2 -14869.134} C_VEL
LIN {X 0,Y 333.29,Z 557.334,A -85,B 0,C 180,E1 -14869.878,E2 -14869.878} C_VEL
LIN {X 0,Y 334.248,Z 546.827,A -85,B 0,C 180,E1 -14870.621,E2 -14870.621} C_VEL
LIN {X 0,Y 335.115,Z 536.496,A -85,B 0,C 180,E1 -14871.168,E2 -14871.168} C_VEL
LIN {X 0,Y 335.754,Z 525.775,A -85,B 0,C 180,E1 -14871.569,E2 -14871.569} C_VEL
LIN {X 0,Y 336.243,Z 502.993,A -85,B 0,C 180,E1 -14872.1,E2 -14872.1} C_VEL
LIN {X 0,Y 337.073,Z 457.454,A -85,B 0,C 180,E1 -14873.071,E2 -14873.071} C_VEL
LIN {X 0,Y 332.456,Z 432.375,A -85,B 0,C 180,E1 -14873.986,E2 -14873.986} C_VEL
LIN {X 0,Y 329.48,Z 418.511,A -85,B 0,C 180,E1 -14874.572,E2 -14874.572} C_VEL
LIN {X 0,Y 329.578,Z 417.044,A -85,B 0,C 180,E1 -14874.941,E2 -14874.941} C_VEL
LIN {X 0,Y 330.214,Z 412.091,A -85,B 0,C 180,E1 -14876.632,E2 -14876.632} C_VEL
LIN {X 0,Y 328.742,Z 403.358,A -85,B 0,C 180,E1 -14879.805,E2 -14879.805} C_VEL
LIN {X 0,Y 326.647,Z 393.403,A -85,B 0,C 180,E1 -14883.588,E2 -14883.588} C_VEL
LIN {X 0,Y 326.63,Z 393.293,A -85,B 0,C 180,E1 -14887.238,E2 -14887.238} C_VEL
LIN {X 0,Y 326.58,Z 393.279,A -85,B 0,C 180,E1 -14891.131,E2 -14891.131} C_VEL
LIN {X 0,Y 326.594,Z 393.299,A -85,B 0,C 180,E1 -14894.754,E2 -14894.754} C_VEL
LIN {X 0,Y 326.631,Z 393.298,A -85,B 0,C 180,E1 -14898.162,E2 -14898.162} C_VEL
LIN {X 0,Y 326.649,Z 393.289,A -85,B 0,C 180,E1 -14901.394,E2 -14901.394} C_VEL
LIN {X 0,Y 326.621,Z 393.289,A -85,B 0,C 180,E1 -14904.85,E2 -14904.85} C_VEL
LIN {X 0,Y 326.616,Z 393.288,A -85,B 0,C 180,E1 -14907.456,E2 -14907.456} C_VEL
LIN {X 0,Y 326.663,Z 393.291,A -85,B 0,C 180,E1 -14910.34,E2 -14910.34} C_VEL
LIN {X 0,Y 326.691,Z 393.274,A -85,B 0,C 180,E1 -14914.516,E2 -14914.516} C_VEL
LIN {X 0,Y 326.646,Z 393.289,A -85,B 0,C 180,E1 -14918.545,E2 -14918.545} C_VEL
LIN {X 0,Y 326.745,Z 393.253,A -85,B 0,C 180,E1 -14921.177,E2 -14921.177} C_VEL
LIN {X 0,Y 326.763,Z 393.278,A -85,B 0,C 180,E1 -14925.432,E2 -14925.432} C_VEL
LIN {X 0,Y 326.769,Z 393.263,A -85,B 0,C 180,E1 -14928.838,E2 -14928.838} C_VEL
LIN {X 0,Y 326.977,Z 393.24,A -85,B 0,C 180,E1 -14932.59,E2 -14932.59} C_VEL
LIN {X 0,Y 326.777,Z 393.278,A -85,B 0,C 180,E1 -14935.064,E2 -14935.064} C_VEL
LIN {X 0,Y 327.046,Z 393.237,A -85,B 0,C 180,E1 -14937.536,E2 -14937.536} C_VEL
LIN {X 0,Y 327.177,Z 393.194,A -85,B 0,C 180,E1 -14939.999,E2 -14939.999} C_VEL
LIN {X 0,Y 327.046,Z 393.232,A -85,B 0,C 180,E1 -14942.463,E2 -14942.463} C_VEL
LIN {X 0,Y 326.969,Z 393.248,A -85,B 0,C 180,E1 -14946.674,E2 -14946.674} C_VEL
LIN {X 0,Y 326.813,Z 393.242,A -85,B 0,C 180,E1 -14949.906,E2 -14949.906} C_VEL
LIN {X 0,Y 326.758,Z 393.281,A -85,B 0,C 180,E1 -14953.685,E2 -14953.685} C_VEL
LIN {X 0,Y 326.696,Z 393.272,A -85,B 0,C 180,E1 -14957.527,E2 -14957.527} C_VEL
LIN {X 0,Y 326.66,Z 393.271,A -85,B 0,C 180,E1 -14960.134,E2 -14960.134} C_VEL
LIN {X 0,Y 326.649,Z 393.294,A -85,B 0,C 180,E1 -14964.128,E2 -14964.128} C_VEL
LIN {X 0,Y 326.68,Z 393.271,A -85,B 0,C 180,E1 -14966.857,E2 -14966.857} C_VEL
LIN {X 0,Y 326.631,Z 393.297,A -85,B 0,C 180,E1 -14970.609,E2 -14970.609} C_VEL
LIN {X 0,Y 326.603,Z 393.283,A -85,B 0,C 180,E1 -14974.019,E2 -14974.019} C_VEL
LIN {X 0,Y 326.626,Z 393.299,A -85,B 0,C 180,E1 -14977.238,E2 -14977.238} C_VEL
LIN {X 0,Y 326.574,Z 393.291,A -85,B 0,C 180,E1 -14981.131,E2 -14981.131} C_VEL
LIN {X 0,Y 326.554,Z 393.302,A -85,B 0,C 180,E1 -14984.748,E2 -14984.748} C_VEL
LIN {X 0,Y 326.577,Z 393.256,A -85,B 0,C 180,E1 -14988.155,E2 -14988.155} C_VEL
LIN {X 0,Y 326.644,Z 393.296,A -85,B 0,C 180,E1 -14991.394,E2 -14991.394} C_VEL
LIN {X 0,Y 326.616,Z 393.271,A -85,B 0,C 180,E1 -14994.851,E2 -14994.851} C_VEL
LIN {X 0,Y 326.604,Z 393.296,A -85,B 0,C 180,E1 -14997.455,E2 -14997.455} C_VEL
LIN {X 0,Y 326.657,Z 393.274,A -85,B 0,C 180,E1 -15000.341,E2 -15000.341} C_VEL
LIN {X 0,Y 326.687,Z 393.293,A -85,B 0,C 180,E1 -15004.516,E2 -15004.516} C_VEL
LIN {X 0,Y 326.692,Z 393.586,A -85,B 0,C 180,E1 -15005.621,E2 -15005.621} C_VEL
LIN {X 0,Y 327.048,Z 394.915,A -85,B 0,C 180,E1 -15005.866,E2 -15005.866} C_VEL
LIN {X 0,Y 328.752,Z 397.552,A -85,B 0,C 180,E1 -15006.209,E2 -15006.209} C_VEL
LIN {X 0,Y 329.922,Z 398.85,A -85,B 0,C 180,E1 -15006.429,E2 -15006.429} C_VEL
LIN {X 0,Y 332.332,Z 402.357,A -85,B 0,C 180,E1 -15006.946,E2 -15006.946} C_VEL
LIN {X 0,Y 333.985,Z 404.384,A -85,B 0,C 180,E1 -15007.285,E2 -15007.285} C_VEL
LIN {X 0,Y 336.998,Z 407.958,A -85,B 0,C 180,E1 -15007.902,E2 -15007.902} C_VEL
LIN {X 0,Y 341.147,Z 412.992,A -85,B 0,C 180,E1 -15008.826,E2 -15008.826} C_VEL
LIN {X 0,Y 343.414,Z 415.457,A -85,B 0,C 180,E1 -15009.321,E2 -15009.321} C_VEL
LIN {X 0,Y 347.347,Z 419.644,A -85,B 0,C 180,E1 -15010.249,E2 -15010.249} C_VEL
LIN {X 0,Y 352.042,Z 424.773,A -85,B 0,C 180,E1 -15011.415,E2 -15011.415} C_VEL
LIN {X 0,Y 354.73,Z 427.231,A -85,B 0,C 180,E1 -15012.089,E2 -15012.089} C_VEL
LIN {X 0,Y 358.928,Z 431.43,A -85,B 0,C 180,E1 -15013.243,E2 -15013.243} C_VEL
LIN {X 0,Y 361.768,Z 433.83,A -85,B 0,C 180,E1 -15014.059,E2 -15014.059} C_VEL
LIN {X 0,Y 365.633,Z 437.699,A -85,B 0,C 180,E1 -15015.257,E2 -15015.257} C_VEL
LIN {X 0,Y 369.613,Z 440.857,A -85,B 0,C 180,E1 -15016.584,E2 -15016.584} C_VEL
LIN {X 0,Y 373.664,Z 444.765,A -85,B 0,C 180,E1 -15018.131,E2 -15018.131} C_VEL
LIN {X 0,Y 377.404,Z 447.22,A -85,B 0,C 180,E1 -15019.711,E2 -15019.711} C_VEL
LIN {X 0,Y 378.642,Z 448.138,A -85,B 0,C 180,E1 -15020.316,E2 -15020.316} C_VEL
LIN {X 0,Y 381.381,Z 451.095,A -85,B 0,C 180,E1 -15021.83,E2 -15021.83} C_VEL
LIN {X 0,Y 383.802,Z 452.967,A -85,B 0,C 180,E1 -15023.391,E2 -15023.391} C_VEL
LIN {X 0,Y 386.149,Z 454.279,A -85,B 0,C 180,E1 -15025.307,E2 -15025.307} C_VEL
LIN {X 0,Y 387.794,Z 454.871,A -85,B 0,C 180,E1 -15027.422,E2 -15027.422} C_VEL
LIN {X 0,Y 388.378,Z 455.295,A -85,B 0,C 180,E1 -15028.963,E2 -15028.963} C_VEL
LIN {X 0,Y 388.542,Z 455.227,A -85,B 0,C 180,E1 -15030,E2 -15030} C_VEL
LIN {X 0,Y 388.258,Z 455.185,A -85,B 0,C 180,E1 -15031.556,E2 -15031.556} C_VEL
LIN {X 0,Y 387.234,Z 454.673,A -85,B 0,C 180,E1 -15033.442,E2 -15033.442} C_VEL
LIN {X 0,Y 385.526,Z 454.003,A -85,B 0,C 180,E1 -15035.229,E2 -15035.229} C_VEL
LIN {X 0,Y 383.279,Z 452.589,A -85,B 0,C 180,E1 -15036.977,E2 -15036.977} C_VEL
LIN {X 0,Y 380.599,Z 450.309,A -85,B 0,C 180,E1 -15038.639,E2 -15038.639} C_VEL
LIN {X 0,Y 377.706,Z 447.351,A -85,B 0,C 180,E1 -15040.146,E2 -15040.146} C_VEL
LIN {X 0,Y 373.851,Z 444.917,A -85,B 0,C 180,E1 -15041.791,E2 -15041.791} C_VEL
LIN {X 0,Y 369.606,Z 440.886,A -85,B 0,C 180,E1 -15043.418,E2 -15043.418} C_VEL
LIN {X 0,Y 367.663,Z 439.253,A -85,B 0,C 180,E1 -15044.071,E2 -15044.071} C_VEL
LIN {X 0,Y 363.712,Z 435.954,A -85,B 0,C 180,E1 -15045.341,E2 -15045.341} C_VEL
LIN {X 0,Y 360.454,Z 432.593,A -85,B 0,C 180,E1 -15046.334,E2 -15046.334} C_VEL
LIN {X 0,Y 356.027,Z 428.685,A -85,B 0,C 180,E1 -15047.557,E2 -15047.557} C_VEL
LIN {X 0,Y 353.162,Z 425.724,A -85,B 0,C 180,E1 -15048.308,E2 -15048.308} C_VEL
LIN {X 0,Y 349.167,Z 421.728,A -85,B 0,C 180,E1 -15049.319,E2 -15049.319} C_VEL
LIN {X 0,Y 346.948,Z 419.308,A -85,B 0,C 180,E1 -15049.841,E2 -15049.841} C_VEL
LIN {X 0,Y 343.169,Z 415.125,A -85,B 0,C 180,E1 -15050.738,E2 -15050.738} C_VEL
LIN {X 0,Y 338.399,Z 409.791,A -85,B 0,C 180,E1 -15051.779,E2 -15051.779} C_VEL
LIN {X 0,Y 336.365,Z 407.356,A -85,B 0,C 180,E1 -15052.228,E2 -15052.228} C_VEL
LIN {X 0,Y 333.429,Z 403.475,A -85,B 0,C 180,E1 -15052.835,E2 -15052.835} C_VEL
LIN {X 0,Y 330.61,Z 400.086,A -85,B 0,C 180,E1 -15053.419,E2 -15053.419} C_VEL
LIN {X 0,Y 329.168,Z 397.933,A -85,B 0,C 180,E1 -15053.716,E2 -15053.716} C_VEL
LIN {X 0,Y 327.33,Z 395.58,A -85,B 0,C 180,E1 -15054.063,E2 -15054.063} C_VEL
LIN {X 0,Y 326.73,Z 393.896,A -85,B 0,C 180,E1 -15054.291,E2 -15054.291} C_VEL
LIN {X 0,Y 326.655,Z 393.331,A -85,B 0,C 180,E1 -15054.635,E2 -15054.635} C_VEL
LIN {X 0,Y 326.651,Z 393.281,A -85,B 0,C 180,E1 -15058.25,E2 -15058.25} C_VEL
LIN {X 0,Y 326.589,Z 393.3,A -85,B 0,C 180,E1 -15061.095,E2 -15061.095} C_VEL
LIN {X 0,Y 326.601,Z 393.274,A -85,B 0,C 180,E1 -15064.019,E2 -15064.019} C_VEL
LIN {X 0,Y 326.627,Z 393.298,A -85,B 0,C 180,E1 -15067.24,E2 -15067.24} C_VEL
LIN {X 0,Y 326.597,Z 393.274,A -85,B 0,C 180,E1 -15070.207,E2 -15070.207} C_VEL
LIN {X 0,Y 326.572,Z 393.27,A -85,B 0,C 180,E1 -15073.523,E2 -15073.523} C_VEL
LIN {X 0,Y 326.606,Z 393.301,A -85,B 0,C 180,E1 -15077.021,E2 -15077.021} C_VEL
LIN {X 0,Y 326.637,Z 393.297,A -85,B 0,C 180,E1 -15081.394,E2 -15081.394} C_VEL
LIN {X 0,Y 326.613,Z 393.282,A -85,B 0,C 180,E1 -15084.851,E2 -15084.851} C_VEL
LIN {X 0,Y 326.601,Z 393.299,A -85,B 0,C 180,E1 -15087.456,E2 -15087.456} C_VEL
LIN {X 0,Y 326.654,Z 393.29,A -85,B 0,C 180,E1 -15090.341,E2 -15090.341} C_VEL
LIN {X 0,Y 326.684,Z 393.281,A -85,B 0,C 180,E1 -15094.517,E2 -15094.517} C_VEL
LIN {X 0,Y 326.639,Z 393.286,A -85,B 0,C 180,E1 -15098.546,E2 -15098.546} C_VEL
LIN {X 0,Y 326.738,Z 393.257,A -85,B 0,C 180,E1 -15101.178,E2 -15101.178} C_VEL
LIN {X 0,Y 326.752,Z 393.282,A -85,B 0,C 180,E1 -15105.28,E2 -15105.28} C_VEL
LIN {X 0,Y 326.102,Z 393.363,A -85,B 0,C 180,E1 -15106.309,E2 -15106.309} C_VEL
LIN {X 0,Y 323.238,Z 393.704,A -85,B 0,C 180,E1 -15107.983,E2 -15107.983} C_VEL
LIN {X 0,Y 320.831,Z 393.99,A -85,B 0,C 180,E1 -15109.34,E2 -15109.34} C_VEL
LIN {X 0,Y 319.846,Z 394.11,A -85,B 0,C 180,E1 -15110.391,E2 -15110.391} C_VEL
LIN {X 0,Y 319.793,Z 394.119,A -85,B 0,C 180,E1 -15110.747,E2 -15110.747} C_VEL
LIN {X 0,Y 319.946,Z 394.127,A -85,B 0,C 180,E1 -15113.695,E2 -15113.695} C_VEL
LIN {X 0,Y 319.987,Z 394.112,A -85,B 0,C 180,E1 -15117.483,E2 -15117.483} C_VEL
LIN {X 0,Y 320.127,Z 394.072,A -85,B 0,C 180,E1 -15120.001,E2 -15120.001} C_VEL
LIN {X 0,Y 319.987,Z 394.117,A -85,B 0,C 180,E1 -15122.518,E2 -15122.518} C_VEL
LIN {X 0,Y 319.947,Z 394.123,A -85,B 0,C 180,E1 -15126.306,E2 -15126.306} C_VEL
LIN {X 0,Y 319.838,Z 394.108,A -85,B 0,C 180,E1 -15128.849,E2 -15128.849} C_VEL
LIN {X 0,Y 319.678,Z 394.16,A -85,B 0,C 180,E1 -15132.701,E2 -15132.701} C_VEL
LIN {X 0,Y 319.696,Z 394.156,A -85,B 0,C 180,E1 -15135.296,E2 -15135.296} C_VEL
LIN {X 0,Y 319.67,Z 394.137,A -85,B 0,C 180,E1 -15139.256,E2 -15139.256} C_VEL
LIN {X 0,Y 319.567,Z 394.175,A -85,B 0,C 180,E1 -15143.32,E2 -15143.32} C_VEL
LIN {X 0,Y 319.632,Z 394.145,A -85,B 0,C 180,E1 -15146.089,E2 -15146.089} C_VEL
LIN {X 0,Y 319.588,Z 394.171,A -85,B 0,C 180,E1 -15148.934,E2 -15148.934} C_VEL
LIN {X 0,Y 319.536,Z 394.178,A -85,B 0,C 180,E1 -15151.862,E2 -15151.862} C_VEL
LIN {X 0,Y 319.578,Z 394.168,A -85,B 0,C 180,E1 -15155.544,E2 -15155.544} C_VEL
LIN {X 0,Y 319.599,Z 394.172,A -85,B 0,C 180,E1 -15158.005,E2 -15158.005} C_VEL
LIN {X 0,Y 319.6,Z 394.172,A -85,B 0,C 180,E1 -15161.613,E2 -15161.613} C_VEL
LIN {X 0,Y 319.586,Z 394.169,A -85,B 0,C 180,E1 -15164.726,E2 -15164.726} C_VEL
LIN {X 0,Y 319.525,Z 394.161,A -85,B 0,C 180,E1 -15168.404,E2 -15168.404} C_VEL
LIN {X 0,Y 319.577,Z 394.176,A -85,B 0,C 180,E1 -15172.345,E2 -15172.345} C_VEL
LIN {X 0,Y 319.617,Z 394.305,A -85,B 0,C 180,E1 -15176.001,E2 -15176.001} C_VEL
LIN {X 0,Y 320.996,Z 400.877,A -85,B 0,C 180,E1 -15178.637,E2 -15178.637} C_VEL
LIN {X 0,Y 322.414,Z 408.168,A -85,B 0,C 180,E1 -15181.344,E2 -15181.344} C_VEL
LIN {X 0,Y 323.172,Z 412.841,A -85,B 0,C 180,E1 -15183.079,E2 -15183.079} C_VEL
LIN {X 0,Y 322.694,Z 417.772,A -85,B 0,C 180,E1 -15184.783,E2 -15184.783} C_VEL
LIN {X 0,Y 322.816,Z 419.101,A -85,B 0,C 180,E1 -15184.925,E2 -15184.925} C_VEL
LIN {X 0,Y 328.437,Z 446.021,A -85,B 0,C 180,E1 -15186.024,E2 -15186.024} C_VEL
LIN {X 0,Y 330.631,Z 459.351,A -85,B 0,C 180,E1 -15186.501,E2 -15186.501} C_VEL
LIN {X 0,Y 329.252,Z 523.002,A -85,B 0,C 180,E1 -15187.901,E2 -15187.901} C_VEL
LIN {X 0,Y 328.745,Z 532.874,A -85,B 0,C 180,E1 -15188.237,E2 -15188.237} C_VEL
LIN {X 0,Y 327.99,Z 542.858,A -85,B 0,C 180,E1 -15188.721,E2 -15188.721} C_VEL
LIN {X 0,Y 326.991,Z 553.211,A -85,B 0,C 180,E1 -15189.394,E2 -15189.394} C_VEL
LIN {X 0,Y 326.035,Z 562.356,A -85,B 0,C 180,E1 -15190.154,E2 -15190.154} C_VEL
LIN {X 0,Y 324.909,Z 571.356,A -85,B 0,C 180,E1 -15191.068,E2 -15191.068} C_VEL
LIN {X 0,Y 323.706,Z 580.081,A -85,B 0,C 180,E1 -15192.142,E2 -15192.142} C_VEL
LIN {X 0,Y 322.703,Z 587.503,A -85,B 0,C 180,E1 -15193.228,E2 -15193.228} C_VEL
LIN {X 0,Y 321.681,Z 595.014,A -85,B 0,C 180,E1 -15194.534,E2 -15194.534} C_VEL
LIN {X 0,Y 320.644,Z 602.293,A -85,B 0,C 180,E1 -15196.049,E2 -15196.049} C_VEL
LIN {X 0,Y 319.629,Z 608.601,A -85,B 0,C 180,E1 -15197.621,E2 -15197.621} C_VEL
LIN {X 0,Y 318.965,Z 613.877,A -85,B 0,C 180,E1 -15199.206,E2 -15199.206} C_VEL
LIN {X 0,Y 318.366,Z 618.972,A -85,B 0,C 180,E1 -15201.111,E2 -15201.111} C_VEL
LIN {X 0,Y 317.99,Z 622.937,A -85,B 0,C 180,E1 -15203.018,E2 -15203.018} C_VEL
LIN {X 0,Y 317.815,Z 625.873,A -85,B 0,C 180,E1 -15204.926,E2 -15204.926} C_VEL
LIN {X 0,Y 317.788,Z 627.375,A -85,B 0,C 180,E1 -15206.196,E2 -15206.196} C_VEL
LIN {X 0,Y 317.734,Z 628.898,A -85,B 0,C 180,E1 -15208.733,E2 -15208.733} C_VEL
LIN {X 0,Y 317.767,Z 629.177,A -85,B 0,C 180,E1 -15210,E2 -15210} C_VEL
LIN {X 0,Y 317.757,Z 628.302,A -85,B 0,C 180,E1 -15212.536,E2 -15212.536} C_VEL
LIN {X 0,Y 317.785,Z 627.374,A -85,B 0,C 180,E1 -15213.805,E2 -15213.805} C_VEL
LIN {X 0,Y 317.827,Z 625.119,A -85,B 0,C 180,E1 -15215.687,E2 -15215.687} C_VEL
LIN {X 0,Y 318.079,Z 621.81,A -85,B 0,C 180,E1 -15217.618,E2 -15217.618} C_VEL
LIN {X 0,Y 318.548,Z 617.455,A -85,B 0,C 180,E1 -15219.525,E2 -15219.525} C_VEL
LIN {X 0,Y 319.201,Z 611.877,A -85,B 0,C 180,E1 -15221.429,E2 -15221.429} C_VEL
LIN {X 0,Y 320.03,Z 606.224,A -85,B 0,C 180,E1 -15223.009,E2 -15223.009} C_VEL
LIN {X 0,Y 321.084,Z 599.421,A -85,B 0,C 180,E1 -15224.579,E2 -15224.579} C_VEL
LIN {X 0,Y 322.175,Z 592.086,A -85,B 0,C 180,E1 -15225.994,E2 -15225.994} C_VEL
LIN {X 0,Y 323.259,Z 583.592,A -85,B 0,C 180,E1 -15227.361,E2 -15227.361} C_VEL
LIN {X 0,Y 324.398,Z 575.289,A -85,B 0,C 180,E1 -15228.472,E2 -15228.472} C_VEL
LIN {X 0,Y 325.64,Z 565.528,A -85,B 0,C 180,E1 -15229.544,E2 -15229.544} C_VEL
LIN {X 0,Y 326.633,Z 557.139,A -85,B 0,C 180,E1 -15230.301,E2 -15230.301} C_VEL
LIN {X 0,Y 327.618,Z 546.632,A -85,B 0,C 180,E1 -15231.058,E2 -15231.058} C_VEL
LIN {X 0,Y 328.509,Z 536.301,A -85,B 0,C 180,E1 -15231.615,E2 -15231.615} C_VEL
LIN {X 0,Y 329.175,Z 525.58,A -85,B 0,C 180,E1 -15232.022,E2 -15232.022} C_VEL
LIN {X 0,Y 329.679,Z 502.798,A -85,B 0,C 180,E1 -15232.564,E2 -15232.564} C_VEL
LIN {X 0,Y 330.54,Z 458.393,A -85,B 0,C 180,E1 -15233.528,E2 -15233.528} C_VEL
LIN {X 0,Y 326.135,Z 434.39,A -85,B 0,C 180,E1 -15234.429,E2 -15234.429} C_VEL
LIN {X 0,Y 322.684,Z 418.34,A -85,B 0,C 180,E1 -15235.122,E2 -15235.122} C_VEL
LIN {X 0,Y 322.812,Z 416.845,A -85,B 0,C 180,E1 -15235.501,E2 -15235.501} C_VEL
LIN {X 0,Y 323.172,Z 412.841,A -85,B 0,C 180,E1 -15236.921,E2 -15236.921} C_VEL
LIN {X 0,Y 321.666,Z 404.163,A -85,B 0,C 180,E1 -15240.167,E2 -15240.167} C_VEL
LIN {X 0,Y 319.623,Z 394.312,A -85,B 0,C 180,E1 -15244.009,E2 -15244.009} C_VEL
LIN {X 0,Y 319.576,Z 394.18,A -85,B 0,C 180,E1 -15248.008,E2 -15248.008} C_VEL
LIN {X 0,Y 319.528,Z 394.16,A -85,B 0,C 180,E1 -15251.597,E2 -15251.597} C_VEL
LIN {X 0,Y 319.589,Z 394.168,A -85,B 0,C 180,E1 -15255.274,E2 -15255.274} C_VEL
LIN {X 0,Y 319.585,Z 394.172,A -85,B 0,C 180,E1 -15258.72,E2 -15258.72} C_VEL
LIN {X 0,Y 319.601,Z 394.175,A -85,B 0,C 180,E1 -15262.338,E2 -15262.338} C_VEL
LIN {X 0,Y 319.562,Z 394.164,A -85,B 0,C 180,E1 -15265.123,E2 -15265.123} C_VEL
LIN {X 0,Y 319.576,Z 394.175,A -85,B 0,C 180,E1 -15269.056,E2 -15269.056} C_VEL
LIN {X 0,Y 319.61,Z 394.15,A -85,B 0,C 180,E1 -15272.498,E2 -15272.498} C_VEL
LIN {X 0,Y 319.605,Z 394.162,A -85,B 0,C 180,E1 -15275.303,E2 -15275.303} C_VEL
LIN {X 0,Y 319.597,Z 394.17,A -85,B 0,C 180,E1 -15278.047,E2 -15278.047} C_VEL
LIN {X 0,Y 319.689,Z 394.133,A -85,B 0,C 180,E1 -15280.962,E2 -15280.962} C_VEL
LIN {X 0,Y 319.731,Z 394.153,A -85,B 0,C 180,E1 -15285.275,E2 -15285.275} C_VEL
LIN {X 0,Y 319.757,Z 394.118,A -85,B 0,C 180,E1 -15289.872,E2 -15289.872} C_VEL
LIN {X 0,Y 319.933,Z 394.112,A -85,B 0,C 180,E1 -15292.426,E2 -15292.426} C_VEL
LIN {X 0,Y 319.746,Z 394.154,A -85,B 0,C 180,E1 -15294.955,E2 -15294.955} C_VEL
LIN {X 0,Y 319.99,Z 394.116,A -85,B 0,C 180,E1 -15297.482,E2 -15297.482} C_VEL
LIN {X 0,Y 320.13,Z 394.071,A -85,B 0,C 180,E1 -15299.999,E2 -15299.999} C_VEL
LIN {X 0,Y 319.99,Z 394.111,A -85,B 0,C 180,E1 -15302.517,E2 -15302.517} C_VEL
LIN {X 0,Y 319.929,Z 394.125,A -85,B 0,C 180,E1 -15306.665,E2 -15306.665} C_VEL
LIN {X 0,Y 319.757,Z 394.12,A -85,B 0,C 180,E1 -15310.126,E2 -15310.126} C_VEL
LIN {X 0,Y 319.729,Z 394.157,A -85,B 0,C 180,E1 -15314.723,E2 -15314.723} C_VEL
LIN {X 0,Y 319.686,Z 394.134,A -85,B 0,C 180,E1 -15319.037,E2 -15319.037} C_VEL
LIN {X 0,Y 319.568,Z 394.179,A -85,B 0,C 180,E1 -15323.319,E2 -15323.319} C_VEL
LIN {X 0,Y 319.631,Z 394.154,A -85,B 0,C 180,E1 -15326.087,E2 -15326.087} C_VEL
LIN {X 0,Y 319.576,Z 394.163,A -85,B 0,C 180,E1 -15328.934,E2 -15328.934} C_VEL
LIN {X 0,Y 319.527,Z 394.182,A -85,B 0,C 180,E1 -15331.861,E2 -15331.861} C_VEL
LIN {X 0,Y 319.577,Z 394.161,A -85,B 0,C 180,E1 -15335.542,E2 -15335.542} C_VEL
LIN {X 0,Y 319.57,Z 394.178,A -85,B 0,C 180,E1 -15338.007,E2 -15338.007} C_VEL
LIN {X 0,Y 319.522,Z 394.172,A -85,B 0,C 180,E1 -15341.597,E2 -15341.597} C_VEL
LIN {X 0,Y 319.512,Z 394.178,A -85,B 0,C 180,E1 -15344.737,E2 -15344.737} C_VEL
LIN {X 0,Y 319.527,Z 394.134,A -85,B 0,C 180,E1 -15348.402,E2 -15348.402} C_VEL
LIN {X 0,Y 319.597,Z 394.176,A -85,B 0,C 180,E1 -15351.996,E2 -15351.996} C_VEL
LIN {X 0,Y 319.557,Z 394.149,A -85,B 0,C 180,E1 -15355.123,E2 -15355.123} C_VEL
LIN {X 0,Y 319.567,Z 394.172,A -85,B 0,C 180,E1 -15359.057,E2 -15359.057} C_VEL
LIN {X 0,Y 319.606,Z 394.171,A -85,B 0,C 180,E1 -15362.498,E2 -15362.498} C_VEL
LIN {X 0,Y 319.676,Z 394.392,A -85,B 0,C 180,E1 -15364.614,E2 -15364.614} C_VEL
LIN {X 0,Y 319.921,Z 395.46,A -85,B 0,C 180,E1 -15364.853,E2 -15364.853} C_VEL
LIN {X 0,Y 321.681,Z 398.339,A -85,B 0,C 180,E1 -15365.19,E2 -15365.19} C_VEL
LIN {X 0,Y 324.765,Z 402.844,A -85,B 0,C 180,E1 -15365.751,E2 -15365.751} C_VEL
LIN {X 0,Y 326.597,Z 405.25,A -85,B 0,C 180,E1 -15366.101,E2 -15366.101} C_VEL
LIN {X 0,Y 330.885,Z 410.691,A -85,B 0,C 180,E1 -15366.944,E2 -15366.944} C_VEL
LIN {X 0,Y 336.262,Z 417.065,A -85,B 0,C 180,E1 -15368.047,E2 -15368.047} C_VEL
LIN {X 0,Y 340.438,Z 421.601,A -85,B 0,C 180,E1 -15368.958,E2 -15368.958} C_VEL
LIN {X 0,Y 344.627,Z 425.86,A -85,B 0,C 180,E1 -15369.901,E2 -15369.901} C_VEL
LIN {X 0,Y 349.572,Z 431.105,A -85,B 0,C 180,E1 -15371.08,E2 -15371.08} C_VEL
LIN {X 0,Y 352.229,Z 433.566,A -85,B 0,C 180,E1 -15371.749,E2 -15371.749} C_VEL
LIN {X 0,Y 356.691,Z 437.885,A -85,B 0,C 180,E1 -15372.934,E2 -15372.934} C_VEL
LIN {X 0,Y 359.645,Z 440.332,A -85,B 0,C 180,E1 -15373.746,E2 -15373.746} C_VEL
LIN {X 0,Y 364.001,Z 444.515,A -85,B 0,C 180,E1 -15375.073,E2 -15375.073} C_VEL
LIN {X 0,Y 367.974,Z 447.694,A -85,B 0,C 180,E1 -15376.368,E2 -15376.368} C_VEL
LIN {X 0,Y 372.203,Z 451.594,A -85,B 0,C 180,E1 -15377.936,E2 -15377.936} C_VEL
LIN {X 0,Y 376.099,Z 454.111,A -85,B 0,C 180,E1 -15379.539,E2 -15379.539} C_VEL
LIN {X 0,Y 377.407,Z 455.144,A -85,B 0,C 180,E1 -15380.169,E2 -15380.169} C_VEL
LIN {X 0,Y 380.162,Z 457.986,A -85,B 0,C 180,E1 -15381.649,E2 -15381.649} C_VEL
LIN {X 0,Y 382.58,Z 459.839,A -85,B 0,C 180,E1 -15383.16,E2 -15383.16} C_VEL
LIN {X 0,Y 384.637,Z 461.027,A -85,B 0,C 180,E1 -15384.758,E2 -15384.758} C_VEL
LIN {X 0,Y 386.062,Z 461.611,A -85,B 0,C 180,E1 -15386.193,E2 -15386.193} C_VEL
LIN {X 0,Y 387.299,Z 462.164,A -85,B 0,C 180,E1 -15388.18,E2 -15388.18} C_VEL
LIN {X 0,Y 387.677,Z 462.274,A -85,B 0,C 180,E1 -15390,E2 -15390} C_VEL
LIN {X 0,Y 387.389,Z 462.232,A -85,B 0,C 180,E1 -15391.559,E2 -15391.559} C_VEL
LIN {X 0,Y 386.607,Z 461.79,A -85,B 0,C 180,E1 -15393.126,E2 -15393.126} C_VEL
LIN {X 0,Y 384.954,Z 461.199,A -85,B 0,C 180,E1 -15394.965,E2 -15394.965} C_VEL
LIN {X 0,Y 382.733,Z 459.937,A -85,B 0,C 180,E1 -15396.733,E2 -15396.733} C_VEL
LIN {X 0,Y 380.026,Z 457.879,A -85,B 0,C 180,E1 -15398.431,E2 -15398.431} C_VEL
LIN {X 0,Y 377.023,Z 454.71,A -85,B 0,C 180,E1 -15400.026,E2 -15400.026} C_VEL
LIN {X 0,Y 372.558,Z 451.83,A -85,B 0,C 180,E1 -15401.931,E2 -15401.931} C_VEL
LIN {X 0,Y 368.163,Z 447.907,A -85,B 0,C 180,E1 -15403.567,E2 -15403.567} C_VEL
LIN {X 0,Y 365.954,Z 445.988,A -85,B 0,C 180,E1 -15404.304,E2 -15404.304} C_VEL
LIN {X 0,Y 361.688,Z 442.506,A -85,B 0,C 180,E1 -15405.631,E2 -15405.631} C_VEL
LIN {X 0,Y 358.084,Z 438.949,A -85,B 0,C 180,E1 -15406.694,E2 -15406.694} C_VEL
LIN {X 0,Y 353.448,Z 434.86,A -85,B 0,C 180,E1 -15407.942,E2 -15407.942} C_VEL
LIN {X 0,Y 349.833,Z 431.313,A -85,B 0,C 180,E1 -15408.856,E2 -15408.856} C_VEL
LIN {X 0,Y 345.707,Z 427.103,A -85,B 0,C 180,E1 -15409.842,E2 -15409.842} C_VEL
LIN {X 0,Y 340.346,Z 421.506,A -85,B 0,C 180,E1 -15411.062,E2 -15411.062} C_VEL
LIN {X 0,Y 334.798,Z 415.23,A -85,B 0,C 180,E1 -15412.261,E2 -15412.261} C_VEL
LIN {X 0,Y 330.05,Z 409.468,A -85,B 0,C 180,E1 -15413.236,E2 -15413.236} C_VEL
LIN {X 0,Y 326.159,Z 404.596,A -85,B 0,C 180,E1 -15413.985,E2 -15413.985} C_VEL
LIN {X 0,Y 322.882,Z 400.228,A -85,B 0,C 180,E1 -15414.598,E2 -15414.598} C_VEL
LIN {X 0,Y 321.437,Z 398.06,A -85,B 0,C 180,E1 -15414.851,E2 -15414.851} C_VEL
LIN {X 0,Y 319.917,Z 395.438,A -85,B 0,C 180,E1 -15415.145,E2 -15415.145} C_VEL
LIN {X 0,Y 319.674,Z 394.38,A -85,B 0,C 180,E1 -15415.385,E2 -15415.385} C_VEL
LIN {X 0,Y 319.584,Z 394.155,A -85,B 0,C 180,E1 -15418.933,E2 -15418.933} C_VEL
LIN {X 0,Y 319.527,Z 394.185,A -85,B 0,C 180,E1 -15421.861,E2 -15421.861} C_VEL
LIN {X 0,Y 319.575,Z 394.151,A -85,B 0,C 180,E1 -15425.543,E2 -15425.543} C_VEL
LIN {X 0,Y 319.595,Z 394.176,A -85,B 0,C 180,E1 -15428.004,E2 -15428.004} C_VEL
LIN {X 0,Y 319.524,Z 394.134,A -85,B 0,C 180,E1 -15431.598,E2 -15431.598} C_VEL
LIN {X 0,Y 319.544,Z 394.175,A -85,B 0,C 180,E1 -15435.268,E2 -15435.268} C_VEL
LIN {X 0,Y 319.539,Z 394.168,A -85,B 0,C 180,E1 -15438.715,E2 -15438.715} C_VEL
LIN {X 0,Y 319.592,Z 394.178,A -85,B 0,C 180,E1 -15442.339,E2 -15442.339} C_VEL
LIN {X 0,Y 319.553,Z 394.159,A -85,B 0,C 180,E1 -15445.124,E2 -15445.124} C_VEL
LIN {X 0,Y 319.564,Z 394.179,A -85,B 0,C 180,E1 -15449.058,E2 -15449.058} C_VEL
LIN {X 0,Y 319.602,Z 394.15,A -85,B 0,C 180,E1 -15452.498,E2 -15452.498} C_VEL
LIN {X 0,Y 319.599,Z 394.172,A -85,B 0,C 180,E1 -15455.304,E2 -15455.304} C_VEL
LIN {X 0,Y 319.59,Z 394.171,A -85,B 0,C 180,E1 -15458.048,E2 -15458.048} C_VEL
LIN {X 0,Y 319.682,Z 394.134,A -85,B 0,C 180,E1 -15460.963,E2 -15460.963} C_VEL
LIN {X 0,Y 319.725,Z 394.157,A -85,B 0,C 180,E1 -15465.276,E2 -15465.276} C_VEL
LIN {X 0,Y 319.753,Z 394.12,A -85,B 0,C 180,E1 -15469.873,E2 -15469.873} C_VEL
LIN {X 0,Y 319.793,Z 394.119,A -85,B 0,C 180,E1 -15470.747,E2 -15470.747} C_VEL
LIN {X 0,Y 319.516,Z 394.164,A -85,B 0,C 180,E1 -15471.45,E2 -15471.45} C_VEL
LIN {X 0,Y 317.545,Z 394.423,A -85,B 0,C 180,E1 -15472.829,E2 -15472.829} C_VEL
LIN {X 0,Y 313.746,Z 394.907,A -85,B 0,C 180,E1 -15474.894,E2 -15474.894} C_VEL
LIN {X 0,Y 312.757,Z 395.025,A -85,B 0,C 180,E1 -15475.969,E2 -15475.969} C_VEL
LIN {X 0,Y 312.719,Z 395.024,A -85,B 0,C 180,E1 -15476.333,E2 -15476.333} C_VEL
LIN {X 0,Y 312.985,Z 394.964,A -85,B 0,C 180,E1 -15478.714,E2 -15478.714} C_VEL
LIN {X 0,Y 312.985,Z 394.976,A -85,B 0,C 180,E1 -15481.287,E2 -15481.287} C_VEL
LIN {X 0,Y 312.714,Z 395.029,A -85,B 0,C 180,E1 -15485.158,E2 -15485.158} C_VEL
LIN {X 0,Y 312.869,Z 394.988,A -85,B 0,C 180,E1 -15487.747,E2 -15487.747} C_VEL
LIN {X 0,Y 312.665,Z 395.022,A -85,B 0,C 180,E1 -15491.672,E2 -15491.672} C_VEL
LIN {X 0,Y 312.696,Z 395.028,A -85,B 0,C 180,E1 -15494.888,E2 -15494.888} C_VEL
LIN {X 0,Y 312.626,Z 395.013,A -85,B 0,C 180,E1 -15499.237,E2 -15499.237} C_VEL
LIN {X 0,Y 312.542,Z 395.051,A -85,B 0,C 180,E1 -15502.79,E2 -15502.79} C_VEL
LIN {X 0,Y 312.6,Z 395.022,A -85,B 0,C 180,E1 -15505.937,E2 -15505.937} C_VEL
LIN {X 0,Y 312.544,Z 395.05,A -85,B 0,C 180,E1 -15509.651,E2 -15509.651} C_VEL
LIN {X 0,Y 312.518,Z 395.036,A -85,B 0,C 180,E1 -15513.69,E2 -15513.69} C_VEL
LIN {X 0,Y 312.552,Z 395.052,A -85,B 0,C 180,E1 -15517.382,E2 -15517.382} C_VEL
LIN {X 0,Y 312.534,Z 395.046,A -85,B 0,C 180,E1 -15520.703,E2 -15520.703} C_VEL
LIN {X 0,Y 312.541,Z 395.045,A -85,B 0,C 180,E1 -15524.195,E2 -15524.195} C_VEL
LIN {X 0,Y 312.486,Z 395.043,A -85,B 0,C 180,E1 -15527.919,E2 -15527.919} C_VEL
LIN {X 0,Y 312.535,Z 395.057,A -85,B 0,C 180,E1 -15531.912,E2 -15531.912} C_VEL
LIN {X 0,Y 312.556,Z 395.208,A -85,B 0,C 180,E1 -15535.553,E2 -15535.553} C_VEL
LIN {X 0,Y 314.074,Z 402.384,A -85,B 0,C 180,E1 -15538.476,E2 -15538.476} C_VEL
LIN {X 0,Y 315.534,Z 409.937,A -85,B 0,C 180,E1 -15541.389,E2 -15541.389} C_VEL
LIN {X 0,Y 316.215,Z 414.673,A -85,B 0,C 180,E1 -15543.192,E2 -15543.192} C_VEL
LIN {X 0,Y 315.93,Z 417.833,A -85,B 0,C 180,E1 -15544.261,E2 -15544.261} C_VEL
LIN {X 0,Y 316.93,Z 422.816,A -85,B 0,C 180,E1 -15544.536,E2 -15544.536} C_VEL
LIN {X 0,Y 322.254,Z 448.905,A -85,B 0,C 180,E1 -15545.608,E2 -15545.608} C_VEL
LIN {X 0,Y 324.116,Z 460.07,A -85,B 0,C 180,E1 -15546.021,E2 -15546.021} C_VEL
LIN {X 0,Y 322.7,Z 522.814,A -85,B 0,C 180,E1 -15547.428,E2 -15547.428} C_VEL
LIN {X 0,Y 322.148,Z 532.679,A -85,B 0,C 180,E1 -15547.768,E2 -15547.768} C_VEL
LIN {X 0,Y 321.36,Z 542.662,A -85,B 0,C 180,E1 -15548.259,E2 -15548.259} C_VEL
LIN {X 0,Y 320.342,Z 553.016,A -85,B 0,C 180,E1 -15548.946,E2 -15548.946} C_VEL
LIN {X 0,Y 319.365,Z 562.161,A -85,B 0,C 180,E1 -15549.721,E2 -15549.721} C_VEL
LIN {X 0,Y 318.202,Z 571.161,A -85,B 0,C 180,E1 -15550.653,E2 -15550.653} C_VEL
LIN {X 0,Y 316.953,Z 579.886,A -85,B 0,C 180,E1 -15551.748,E2 -15551.748} C_VEL
LIN {X 0,Y 315.899,Z 587.308,A -85,B 0,C 180,E1 -15552.856,E2 -15552.856} C_VEL
LIN {X 0,Y 314.603,Z 596.105,A -85,B 0,C 180,E1 -15554.451,E2 -15554.451} C_VEL
LIN {X 0,Y 313.723,Z 602.097,A -85,B 0,C 180,E1 -15555.735,E2 -15555.735} C_VEL
LIN {X 0,Y 312.67,Z 608.405,A -85,B 0,C 180,E1 -15557.341,E2 -15557.341} C_VEL
LIN {X 0,Y 311.962,Z 613.681,A -85,B 0,C 180,E1 -15558.961,E2 -15558.961} C_VEL
LIN {X 0,Y 311.313,Z 618.776,A -85,B 0,C 180,E1 -15560.908,E2 -15560.908} C_VEL
LIN {X 0,Y 310.922,Z 622.742,A -85,B 0,C 180,E1 -15562.859,E2 -15562.859} C_VEL
LIN {X 0,Y 310.721,Z 625.677,A -85,B 0,C 180,E1 -15564.81,E2 -15564.81} C_VEL
LIN {X 0,Y 310.701,Z 627.179,A -85,B 0,C 180,E1 -15566.109,E2 -15566.109} C_VEL
LIN {X 0,Y 310.649,Z 628.703,A -85,B 0,C 180,E1 -15568.704,E2 -15568.704} C_VEL
LIN {X 0,Y 310.678,Z 628.983,A -85,B 0,C 180,E1 -15570,E2 -15570} C_VEL
LIN {X 0,Y 310.679,Z 628.107,A -85,B 0,C 180,E1 -15572.593,E2 -15572.593} C_VEL
LIN {X 0,Y 310.698,Z 627.179,A -85,B 0,C 180,E1 -15573.891,E2 -15573.891} C_VEL
LIN {X 0,Y 310.726,Z 625.174,A -85,B 0,C 180,E1 -15575.616,E2 -15575.616} C_VEL
LIN {X 0,Y 311.021,Z 621.615,A -85,B 0,C 180,E1 -15577.792,E2 -15577.792} C_VEL
LIN {X 0,Y 311.503,Z 617.259,A -85,B 0,C 180,E1 -15579.742,E2 -15579.742} C_VEL
LIN {X 0,Y 312.195,Z 611.68,A -85,B 0,C 180,E1 -15581.69,E2 -15581.69} C_VEL
LIN {X 0,Y 313.104,Z 606.029,A -85,B 0,C 180,E1 -15583.302,E2 -15583.302} C_VEL
LIN {X 0,Y 314.178,Z 599.225,A -85,B 0,C 180,E1 -15584.907,E2 -15584.907} C_VEL
LIN {X 0,Y 315.397,Z 591.336,A -85,B 0,C 180,E1 -15586.447,E2 -15586.447} C_VEL
LIN {X 0,Y 316.495,Z 583.177,A -85,B 0,C 180,E1 -15587.778,E2 -15587.778} C_VEL
LIN {X 0,Y 317.673,Z 575.094,A -85,B 0,C 180,E1 -15588.878,E2 -15588.878} C_VEL
LIN {X 0,Y 318.949,Z 565.333,A -85,B 0,C 180,E1 -15589.971,E2 -15589.971} C_VEL
LIN {X 0,Y 319.993,Z 556.944,A -85,B 0,C 180,E1 -15590.742,E2 -15590.742} C_VEL
LIN {X 0,Y 321.009,Z 546.437,A -85,B 0,C 180,E1 -15591.513,E2 -15591.513} C_VEL
LIN {X 0,Y 321.93,Z 536.106,A -85,B 0,C 180,E1 -15592.08,E2 -15592.08} C_VEL
LIN {X 0,Y 322.62,Z 525.386,A -85,B 0,C 180,E1 -15592.494,E2 -15592.494} C_VEL
LIN {X 0,Y 323.216,Z 501.257,A -85,B 0,C 180,E1 -15593.073,E2 -15593.073} C_VEL
LIN {X 0,Y 324.093,Z 459.683,A -85,B 0,C 180,E1 -15593.99,E2 -15593.99} C_VEL
LIN {X 0,Y 319.68,Z 435.55,A -85,B 0,C 180,E1 -15594.923,E2 -15594.923} C_VEL
LIN {X 0,Y 315.933,Z 418.168,A -85,B 0,C 180,E1 -15595.695,E2 -15595.695} C_VEL
LIN {X 0,Y 316.013,Z 416.739,A -85,B 0,C 180,E1 -15596.055,E2 -15596.055} C_VEL
LIN {X 0,Y 316.163,Z 413.542,A -85,B 0,C 180,E1 -15597.231,E2 -15597.231} C_VEL
LIN {X 0,Y 314.603,Z 404.965,A -85,B 0,C 180,E1 -15600.547,E2 -15600.547} C_VEL
LIN {X 0,Y 312.699,Z 395.816,A -85,B 0,C 180,E1 -15604.186,E2 -15604.186} C_VEL
LIN {X 0,Y 312.549,Z 395.116,A -85,B 0,C 180,E1 -15604.595,E2 -15604.595} C_VEL
LIN {X 0,Y 312.537,Z 395.057,A -85,B 0,C 180,E1 -15608.089,E2 -15608.089} C_VEL
LIN {X 0,Y 312.489,Z 395.042,A -85,B 0,C 180,E1 -15612.081,E2 -15612.081} C_VEL
LIN {X 0,Y 312.549,Z 395.044,A -85,B 0,C 180,E1 -15616.017,E2 -15616.017} C_VEL
LIN {X 0,Y 312.549,Z 395.04,A -85,B 0,C 180,E1 -15619.865,E2 -15619.865} C_VEL
LIN {X 0,Y 312.555,Z 395.051,A -85,B 0,C 180,E1 -15622.618,E2 -15622.618} C_VEL
LIN {X 0,Y 312.521,Z 395.036,A -85,B 0,C 180,E1 -15626.31,E2 -15626.31} C_VEL
LIN {X 0,Y 312.548,Z 395.049,A -85,B 0,C 180,E1 -15630.35,E2 -15630.35} C_VEL
LIN {X 0,Y 312.603,Z 395.021,A -85,B 0,C 180,E1 -15634.064,E2 -15634.064} C_VEL
LIN {X 0,Y 312.588,Z 395.047,A -85,B 0,C 180,E1 -15637.528,E2 -15637.528} C_VEL
LIN {X 0,Y 312.638,Z 395.008,A -85,B 0,C 180,E1 -15641.656,E2 -15641.656} C_VEL
LIN {X 0,Y 312.694,Z 395.033,A -85,B 0,C 180,E1 -15645.685,E2 -15645.685} C_VEL
LIN {X 0,Y 312.701,Z 394.998,A -85,B 0,C 180,E1 -15649.641,E2 -15649.641} C_VEL
LIN {X 0,Y 312.873,Z 394.987,A -85,B 0,C 180,E1 -15652.254,E2 -15652.254} C_VEL
LIN {X 0,Y 312.717,Z 395.029,A -85,B 0,C 180,E1 -15654.842,E2 -15654.842} C_VEL
LIN {X 0,Y 312.989,Z 394.976,A -85,B 0,C 180,E1 -15658.713,E2 -15658.713} C_VEL
LIN {X 0,Y 312.987,Z 394.964,A -85,B 0,C 180,E1 -15661.286,E2 -15661.286} C_VEL
LIN {X 0,Y 312.717,Z 395.031,A -85,B 0,C 180,E1 -15665.157,E2 -15665.157} C_VEL
LIN {X 0,Y 312.87,Z 394.997,A -85,B 0,C 180,E1 -15667.745,E2 -15667.745} C_VEL
LIN {X 0,Y 312.67,Z 395.013,A -85,B 0,C 180,E1 -15671.671,E2 -15671.671} C_VEL
LIN {X 0,Y 312.698,Z 395.033,A -85,B 0,C 180,E1 -15674.887,E2 -15674.887} C_VEL
LIN {X 0,Y 312.627,Z 395.012,A -85,B 0,C 180,E1 -15679.235,E2 -15679.235} C_VEL
LIN {X 0,Y 312.543,Z 395.051,A -85,B 0,C 180,E1 -15682.789,E2 -15682.789} C_VEL
LIN {X 0,Y 312.599,Z 395.031,A -85,B 0,C 180,E1 -15685.935,E2 -15685.935} C_VEL
LIN {X 0,Y 312.535,Z 395.047,A -85,B 0,C 180,E1 -15689.65,E2 -15689.65} C_VEL
LIN {X 0,Y 312.516,Z 395.039,A -85,B 0,C 180,E1 -15693.688,E2 -15693.688} C_VEL
LIN {X 0,Y 312.535,Z 395.056,A -85,B 0,C 180,E1 -15697.383,E2 -15697.383} C_VEL
LIN {X 0,Y 312.486,Z 395.044,A -85,B 0,C 180,E1 -15700.709,E2 -15700.709} C_VEL
LIN {X 0,Y 312.47,Z 395.06,A -85,B 0,C 180,E1 -15704.205,E2 -15704.205} C_VEL
LIN {X 0,Y 312.485,Z 395.009,A -85,B 0,C 180,E1 -15707.917,E2 -15707.917} C_VEL
LIN {X 0,Y 312.555,Z 395.054,A -85,B 0,C 180,E1 -15711.904,E2 -15711.904} C_VEL
LIN {X 0,Y 312.503,Z 395.027,A -85,B 0,C 180,E1 -15715.79,E2 -15715.79} C_VEL
LIN {X 0,Y 312.52,Z 395.052,A -85,B 0,C 180,E1 -15718.854,E2 -15718.854} C_VEL
LIN {X 0,Y 312.571,Z 395.035,A -85,B 0,C 180,E1 -15721.824,E2 -15721.824} C_VEL
LIN {X 0,Y 312.604,Z 395.218,A -85,B 0,C 180,E1 -15723.741,E2 -15723.741} C_VEL
LIN {X 0,Y 312.825,Z 396.108,A -85,B 0,C 180,E1 -15723.979,E2 -15723.979} C_VEL
LIN {X 0,Y 314.29,Z 398.84,A -85,B 0,C 180,E1 -15724.258,E2 -15724.258} C_VEL
LIN {X 0,Y 317.385,Z 403.463,A -85,B 0,C 180,E1 -15724.753,E2 -15724.753} C_VEL
LIN {X 0,Y 320.824,Z 408.323,A -85,B 0,C 180,E1 -15725.35,E2 -15725.35} C_VEL
LIN {X 0,Y 325.426,Z 413.929,A -85,B 0,C 180,E1 -15726.171,E2 -15726.171} C_VEL
LIN {X 0,Y 329.994,Z 419.321,A -85,B 0,C 180,E1 -15727.046,E2 -15727.046} C_VEL
LIN {X 0,Y 335.058,Z 425.05,A -85,B 0,C 180,E1 -15728.074,E2 -15728.074} C_VEL
LIN {X 0,Y 341.132,Z 431.401,A -85,B 0,C 180,E1 -15729.382,E2 -15729.382} C_VEL
LIN {X 0,Y 347.399,Z 437.74,A -85,B 0,C 180,E1 -15730.834,E2 -15730.834} C_VEL
LIN {X 0,Y 354.223,Z 444.134,A -85,B 0,C 180,E1 -15732.558,E2 -15732.558} C_VEL
LIN {X 0,Y 357.704,Z 447.092,A -85,B 0,C 180,E1 -15733.505,E2 -15733.505} C_VEL
LIN {X 0,Y 362.192,Z 451.215,A -85,B 0,C 180,E1 -15734.832,E2 -15734.832} C_VEL
LIN {X 0,Y 366.013,Z 454.222,A -85,B 0,C 180,E1 -15736.053,E2 -15736.053} C_VEL
LIN {X 0,Y 370.189,Z 458.027,A -85,B 0,C 180,E1 -15737.548,E2 -15737.548} C_VEL
LIN {X 0,Y 374.311,Z 460.747,A -85,B 0,C 180,E1 -15739.178,E2 -15739.178} C_VEL
LIN {X 0,Y 375.881,Z 461.799,A -85,B 0,C 180,E1 -15739.874,E2 -15739.874} C_VEL
LIN {X 0,Y 378.947,Z 464.876,A -85,B 0,C 180,E1 -15741.467,E2 -15741.467} C_VEL
LIN {X 0,Y 381.669,Z 466.904,A -85,B 0,C 180,E1 -15743.143,E2 -15743.143} C_VEL
LIN {X 0,Y 384.063,Z 468.238,A -85,B 0,C 180,E1 -15745.023,E2 -15745.023} C_VEL
LIN {X 0,Y 385.733,Z 468.806,A -85,B 0,C 180,E1 -15746.866,E2 -15746.866} C_VEL
LIN {X 0,Y 386.655,Z 469.383,A -85,B 0,C 180,E1 -15748.958,E2 -15748.958} C_VEL
LIN {X 0,Y 386.811,Z 469.321,A -85,B 0,C 180,E1 -15750,E2 -15750} C_VEL
LIN {X 0,Y 386.523,Z 469.257,A -85,B 0,C 180,E1 -15751.563,E2 -15751.563} C_VEL
LIN {X 0,Y 385.729,Z 468.836,A -85,B 0,C 180,E1 -15753.133,E2 -15753.133} C_VEL
LIN {X 0,Y 384.063,Z 468.249,A -85,B 0,C 180,E1 -15754.977,E2 -15754.977} C_VEL
LIN {X 0,Y 381.667,Z 466.906,A -85,B 0,C 180,E1 -15756.858,E2 -15756.858} C_VEL
LIN {X 0,Y 378.693,Z 464.649,A -85,B 0,C 180,E1 -15758.683,E2 -15758.683} C_VEL
LIN {X 0,Y 375.162,Z 461.143,A -85,B 0,C 180,E1 -15760.465,E2 -15760.465} C_VEL
LIN {X 0,Y 371.14,Z 458.733,A -85,B 0,C 180,E1 -15762.099,E2 -15762.099} C_VEL
LIN {X 0,Y 366.628,Z 454.832,A -85,B 0,C 180,E1 -15763.741,E2 -15763.741} C_VEL
LIN {X 0,Y 363.842,Z 452.451,A -85,B 0,C 180,E1 -15764.66,E2 -15764.66} C_VEL
LIN {X 0,Y 358.945,Z 448.37,A -85,B 0,C 180,E1 -15766.135,E2 -15766.135} C_VEL
LIN {X 0,Y 355.26,Z 444.948,A -85,B 0,C 180,E1 -15767.162,E2 -15767.162} C_VEL
LIN {X 0,Y 350.484,Z 440.726,A -85,B 0,C 180,E1 -15768.394,E2 -15768.394} C_VEL
LIN {X 0,Y 346.815,Z 437.21,A -85,B 0,C 180,E1 -15769.303,E2 -15769.303} C_VEL
LIN {X 0,Y 342.182,Z 432.378,A -85,B 0,C 180,E1 -15770.385,E2 -15770.385} C_VEL
LIN {X 0,Y 336.961,Z 427.148,A -85,B 0,C 180,E1 -15771.513,E2 -15771.513} C_VEL
LIN {X 0,Y 331.057,Z 420.612,A -85,B 0,C 180,E1 -15772.734,E2 -15772.734} C_VEL
LIN {X 0,Y 326.219,Z 414.861,A -85,B 0,C 180,E1 -15773.679,E2 -15773.679} C_VEL
LIN {X 0,Y 322.174,Z 409.968,A -85,B 0,C 180,E1 -15774.422,E2 -15774.422} C_VEL
LIN {X 0,Y 318.203,Z 404.749,A -85,B 0,C 180,E1 -15775.105,E2 -15775.105} C_VEL
LIN {X 0,Y 314.997,Z 399.873,A -85,B 0,C 180,E1 -15775.63,E2 -15775.63} C_VEL
LIN {X 0,Y 312.908,Z 396.408,A -85,B 0,C 180,E1 -15775.986,E2 -15775.986} C_VEL
LIN {X 0,Y 312.617,Z 395.337,A -85,B 0,C 180,E1 -15776.194,E2 -15776.194} C_VEL
LIN {X 0,Y 312.55,Z 395.054,A -85,B 0,C 180,E1 -15776.725,E2 -15776.725} C_VEL
LIN {X 0,Y 312.54,Z 395.032,A -85,B 0,C 180,E1 -15779.65,E2 -15779.65} C_VEL
LIN {X 0,Y 312.513,Z 395.03,A -85,B 0,C 180,E1 -15783.689,E2 -15783.689} C_VEL
LIN {X 0,Y 312.548,Z 395.054,A -85,B 0,C 180,E1 -15787.381,E2 -15787.381} C_VEL
LIN {X 0,Y 312.489,Z 395.019,A -85,B 0,C 180,E1 -15790.708,E2 -15790.708} C_VEL
LIN {X 0,Y 312.47,Z 395.039,A -85,B 0,C 180,E1 -15794.205,E2 -15794.205} C_VEL
LIN {X 0,Y 312.525,Z 395.05,A -85,B 0,C 180,E1 -15797.909,E2 -15797.909} C_VEL
LIN {X 0,Y 312.55,Z 395.052,A -85,B 0,C 180,E1 -15801.905,E2 -15801.905} C_VEL
LIN {X 0,Y 312.499,Z 395.038,A -85,B 0,C 180,E1 -15805.79,E2 -15805.79} C_VEL
LIN {X 0,Y 312.517,Z 395.058,A -85,B 0,C 180,E1 -15808.854,E2 -15808.854} C_VEL
LIN {X 0,Y 312.568,Z 395.029,A -85,B 0,C 180,E1 -15811.825,E2 -15811.825} C_VEL
LIN {X 0,Y 312.579,Z 395.04,A -85,B 0,C 180,E1 -15814.711,E2 -15814.711} C_VEL
LIN {X 0,Y 312.581,Z 395.045,A -85,B 0,C 180,E1 -15817.529,E2 -15817.529} C_VEL
LIN {X 0,Y 312.632,Z 395.016,A -85,B 0,C 180,E1 -15821.657,E2 -15821.657} C_VEL
LIN {X 0,Y 312.688,Z 395.034,A -85,B 0,C 180,E1 -15825.687,E2 -15825.687} C_VEL
LIN {X 0,Y 312.697,Z 394.999,A -85,B 0,C 180,E1 -15829.642,E2 -15829.642} C_VEL
LIN {X 0,Y 312.866,Z 394.998,A -85,B 0,C 180,E1 -15832.255,E2 -15832.255} C_VEL
LIN {X 0,Y 312.714,Z 395.031,A -85,B 0,C 180,E1 -15834.843,E2 -15834.843} C_VEL
LIN {X 0,Y 312.719,Z 395.024,A -85,B 0,C 180,E1 -15836.333,E2 -15836.333} C_VEL
LIN {X 0,Y 312.187,Z 395.083,A -85,B 0,C 180,E1 -15837.411,E2 -15837.411} C_VEL
LIN {X 0,Y 309.452,Z 395.409,A -85,B 0,C 180,E1 -15839.169,E2 -15839.169} C_VEL
LIN {X 0,Y 307.047,Z 395.709,A -85,B 0,C 180,E1 -15840.594,E2 -15840.594} C_VEL
LIN {X 0,Y 305.989,Z 395.852,A -85,B 0,C 180,E1 -15841.696,E2 -15841.696} C_VEL
LIN {X 0,Y 305.892,Z 395.865,A -85,B 0,C 180,E1 -15842.07,E2 -15842.07} C_VEL
LIN {X 0,Y 305.848,Z 395.876,A -85,B 0,C 180,E1 -15846.598,E2 -15846.598} C_VEL
LIN {X 0,Y 305.731,Z 395.862,A -85,B 0,C 180,E1 -15849.261,E2 -15849.261} C_VEL
LIN {X 0,Y 305.584,Z 395.915,A -85,B 0,C 180,E1 -15853.297,E2 -15853.297} C_VEL
LIN {X 0,Y 305.59,Z 395.906,A -85,B 0,C 180,E1 -15856.021,E2 -15856.021} C_VEL
LIN {X 0,Y 305.573,Z 395.893,A -85,B 0,C 180,E1 -15859.446,E2 -15859.446} C_VEL
LIN {X 0,Y 305.487,Z 395.929,A -85,B 0,C 180,E1 -15863.042,E2 -15863.042} C_VEL
LIN {X 0,Y 305.545,Z 395.898,A -85,B 0,C 180,E1 -15866.228,E2 -15866.228} C_VEL
LIN {X 0,Y 305.495,Z 395.926,A -85,B 0,C 180,E1 -15869.051,E2 -15869.051} C_VEL
LIN {X 0,Y 305.446,Z 395.931,A -85,B 0,C 180,E1 -15871.953,E2 -15871.953} C_VEL
LIN {X 0,Y 305.461,Z 395.922,A -85,B 0,C 180,E1 -15875.114,E2 -15875.114} C_VEL
LIN {X 0,Y 305.492,Z 395.924,A -85,B 0,C 180,E1 -15878.54,E2 -15878.54} C_VEL
LIN {X 0,Y 305.514,Z 395.928,A -85,B 0,C 180,E1 -15882.599,E2 -15882.599} C_VEL
LIN {X 0,Y 305.467,Z 395.936,A -85,B 0,C 180,E1 -15886.354,E2 -15886.354} C_VEL
LIN {X 0,Y 305.458,Z 395.909,A -85,B 0,C 180,E1 -15889.893,E2 -15889.893} C_VEL
LIN {X 0,Y 305.484,Z 395.916,A -85,B 0,C 180,E1 -15893.632,E2 -15893.632} C_VEL
LIN {X 0,Y 305.515,Z 396.04,A -85,B 0,C 180,E1 -15895.042,E2 -15895.042} C_VEL
LIN {X 0,Y 307.146,Z 403.728,A -85,B 0,C 180,E1 -15898.247,E2 -15898.247} C_VEL
LIN {X 0,Y 308.367,Z 410.017,A -85,B 0,C 180,E1 -15900.771,E2 -15900.771} C_VEL
LIN {X 0,Y 309.243,Z 415.59,A -85,B 0,C 180,E1 -15902.966,E2 -15902.966} C_VEL
LIN {X 0,Y 309.144,Z 417.77,A -85,B 0,C 180,E1 -15903.675,E2 -15903.675} C_VEL
LIN {X 0,Y 311.72,Z 429.441,A -85,B 0,C 180,E1 -15904.249,E2 -15904.249} C_VEL
LIN {X 0,Y 316.387,Z 453.516,A -85,B 0,C 180,E1 -15905.242,E2 -15905.242} C_VEL
LIN {X 0,Y 317.631,Z 461.617,A -85,B 0,C 180,E1 -15905.542,E2 -15905.542} C_VEL
LIN {X 0,Y 316.166,Z 522.626,A -85,B 0,C 180,E1 -15906.935,E2 -15906.935} C_VEL
LIN {X 0,Y 315.6,Z 532.484,A -85,B 0,C 180,E1 -15907.281,E2 -15907.281} C_VEL
LIN {X 0,Y 314.782,Z 542.467,A -85,B 0,C 180,E1 -15907.781,E2 -15907.781} C_VEL
LIN {X 0,Y 313.743,Z 552.821,A -85,B 0,C 180,E1 -15908.482,E2 -15908.482} C_VEL
LIN {X 0,Y 312.719,Z 561.966,A -85,B 0,C 180,E1 -15909.271,E2 -15909.271} C_VEL
LIN {X 0,Y 311.482,Z 570.965,A -85,B 0,C 180,E1 -15910.218,E2 -15910.218} C_VEL
LIN {X 0,Y 310.192,Z 579.69,A -85,B 0,C 180,E1 -15911.336,E2 -15911.336} C_VEL
LIN {X 0,Y 309.092,Z 587.112,A -85,B 0,C 180,E1 -15912.467,E2 -15912.467} C_VEL
LIN {X 0,Y 307.758,Z 595.91,A -85,B 0,C 180,E1 -15914.096,E2 -15914.096} C_VEL
LIN {X 0,Y 306.815,Z 601.901,A -85,B 0,C 180,E1 -15915.407,E2 -15915.407} C_VEL
LIN {X 0,Y 305.732,Z 608.21,A -85,B 0,C 180,E1 -15917.049,E2 -15917.049} C_VEL
LIN {X 0,Y 304.967,Z 613.485,A -85,B 0,C 180,E1 -15918.704,E2 -15918.704} C_VEL
LIN {X 0,Y 304.272,Z 618.58,A -85,B 0,C 180,E1 -15920.696,E2 -15920.696} C_VEL
LIN {X 0,Y 303.843,Z 622.545,A -85,B 0,C 180,E1 -15922.692,E2 -15922.692} C_VEL
LIN {X 0,Y 303.64,Z 625.482,A -85,B 0,C 180,E1 -15924.688,E2 -15924.688} C_VEL
LIN {X 0,Y 303.598,Z 626.984,A -85,B 0,C 180,E1 -15926.018,E2 -15926.018} C_VEL
LIN {X 0,Y 303.566,Z 628.508,A -85,B 0,C 180,E1 -15928.674,E2 -15928.674} C_VEL
LIN {X 0,Y 303.591,Z 628.788,A -85,B 0,C 180,E1 -15930,E2 -15930} C_VEL
LIN {X 0,Y 303.603,Z 627.913,A -85,B 0,C 180,E1 -15932.654,E2 -15932.654} C_VEL
LIN {X 0,Y 303.593,Z 626.983,A -85,B 0,C 180,E1 -15933.983,E2 -15933.983} C_VEL
LIN {X 0,Y 303.741,Z 623.633,A -85,B 0,C 180,E1 -15936.644,E2 -15936.644} C_VEL
LIN {X 0,Y 304.116,Z 620.007,A -85,B 0,C 180,E1 -15938.64,E2 -15938.64} C_VEL
LIN {X 0,Y 304.698,Z 615.273,A -85,B 0,C 180,E1 -15940.634,E2 -15940.634} C_VEL
LIN {X 0,Y 305.389,Z 610.392,A -85,B 0,C 180,E1 -15942.291,E2 -15942.291} C_VEL
LIN {X 0,Y 306.356,Z 604.521,A -85,B 0,C 180,E1 -15943.938,E2 -15943.938} C_VEL
LIN {X 0,Y 307.273,Z 599.028,A -85,B 0,C 180,E1 -15945.25,E2 -15945.25} C_VEL
LIN {X 0,Y 308.457,Z 591.893,A -85,B 0,C 180,E1 -15946.689,E2 -15946.689} C_VEL
LIN {X 0,Y 309.704,Z 582.981,A -85,B 0,C 180,E1 -15948.181,E2 -15948.181} C_VEL
LIN {X 0,Y 310.945,Z 574.898,A -85,B 0,C 180,E1 -15949.303,E2 -15949.303} C_VEL
LIN {X 0,Y 312.27,Z 565.137,A -85,B 0,C 180,E1 -15950.417,E2 -15950.417} C_VEL
LIN {X 0,Y 313.362,Z 556.749,A -85,B 0,C 180,E1 -15951.201,E2 -15951.201} C_VEL
LIN {X 0,Y 314.424,Z 546.242,A -85,B 0,C 180,E1 -15951.987,E2 -15951.987} C_VEL
LIN {X 0,Y 315.349,Z 535.911,A -85,B 0,C 180,E1 -15952.566,E2 -15952.566} C_VEL
LIN {X 0,Y 316.086,Z 525.191,A -85,B 0,C 180,E1 -15952.985,E2 -15952.985} C_VEL
LIN {X 0,Y 316.694,Z 501.229,A -85,B 0,C 180,E1 -15953.573,E2 -15953.573} C_VEL
LIN {X 0,Y 317.498,Z 459.847,A -85,B 0,C 180,E1 -15954.512,E2 -15954.512} C_VEL
LIN {X 0,Y 312.984,Z 435.468,A -85,B 0,C 180,E1 -15955.491,E2 -15955.491} C_VEL
LIN {X 0,Y 309.163,Z 418,A -85,B 0,C 180,E1 -15956.297,E2 -15956.297} C_VEL
LIN {X 0,Y 309.221,Z 416.538,A -85,B 0,C 180,E1 -15956.672,E2 -15956.672} C_VEL
LIN {X 0,Y 308.671,Z 411.704,A -85,B 0,C 180,E1 -15958.564,E2 -15958.564} C_VEL
LIN {X 0,Y 306.948,Z 402.908,A -85,B 0,C 180,E1 -15962.094,E2 -15962.094} C_VEL
LIN {X 0,Y 305.521,Z 396.022,A -85,B 0,C 180,E1 -15964.972,E2 -15964.972} C_VEL
LIN {X 0,Y 305.469,Z 395.933,A -85,B 0,C 180,E1 -15968.532,E2 -15968.532} C_VEL
LIN {X 0,Y 305.465,Z 395.924,A -85,B 0,C 180,E1 -15972.587,E2 -15972.587} C_VEL
LIN {X 0,Y 305.503,Z 395.924,A -85,B 0,C 180,E1 -15976.358,E2 -15976.358} C_VEL
LIN {X 0,Y 305.502,Z 395.917,A -85,B 0,C 180,E1 -15979.898,E2 -15979.898} C_VEL
LIN {X 0,Y 305.504,Z 395.929,A -85,B 0,C 180,E1 -15983.625,E2 -15983.625} C_VEL
LIN {X 0,Y 305.467,Z 395.915,A -85,B 0,C 180,E1 -15986.483,E2 -15986.483} C_VEL
LIN {X 0,Y 305.468,Z 395.936,A -85,B 0,C 180,E1 -15989.591,E2 -15989.591} C_VEL
LIN {X 0,Y 305.522,Z 395.902,A -85,B 0,C 180,E1 -15992.608,E2 -15992.608} C_VEL
LIN {X 0,Y 305.509,Z 395.919,A -85,B 0,C 180,E1 -15995.538,E2 -15995.538} C_VEL
LIN {X 0,Y 305.519,Z 395.907,A -85,B 0,C 180,E1 -15999.814,E2 -15999.814} C_VEL
LIN {X 0,Y 305.575,Z 395.894,A -85,B 0,C 180,E1 -16002.602,E2 -16002.602} C_VEL
LIN {X 0,Y 305.649,Z 395.907,A -85,B 0,C 180,E1 -16005.348,E2 -16005.348} C_VEL
LIN {X 0,Y 305.638,Z 395.88,A -85,B 0,C 180,E1 -16009.399,E2 -16009.399} C_VEL
LIN {X 0,Y 305.814,Z 395.862,A -85,B 0,C 180,E1 -16012.074,E2 -16012.074} C_VEL
LIN {X 0,Y 305.688,Z 395.905,A -85,B 0,C 180,E1 -16014.723,E2 -16014.723} C_VEL
LIN {X 0,Y 305.956,Z 395.851,A -85,B 0,C 180,E1 -16018.683,E2 -16018.683} C_VEL
LIN {X 0,Y 305.954,Z 395.839,A -85,B 0,C 180,E1 -16021.315,E2 -16021.315} C_VEL
LIN {X 0,Y 305.688,Z 395.907,A -85,B 0,C 180,E1 -16025.276,E2 -16025.276} C_VEL
LIN {X 0,Y 305.811,Z 395.874,A -85,B 0,C 180,E1 -16027.925,E2 -16027.925} C_VEL
LIN {X 0,Y 305.604,Z 395.897,A -85,B 0,C 180,E1 -16031.944,E2 -16031.944} C_VEL
LIN {X 0,Y 305.636,Z 395.914,A -85,B 0,C 180,E1 -16035.034,E2 -16035.034} C_VEL
LIN {X 0,Y 305.574,Z 395.89,A -85,B 0,C 180,E1 -16039.444,E2 -16039.444} C_VEL
LIN {X 0,Y 305.488,Z 395.931,A -85,B 0,C 180,E1 -16043.041,E2 -16043.041} C_VEL
LIN {X 0,Y 305.528,Z 395.91,A -85,B 0,C 180,E1 -16046.22,E2 -16046.22} C_VEL
LIN {X 0,Y 305.485,Z 395.919,A -85,B 0,C 180,E1 -16049.047,E2 -16049.047} C_VEL
LIN {X 0,Y 305.439,Z 395.936,A -85,B 0,C 180,E1 -16051.952,E2 -16051.952} C_VEL
LIN {X 0,Y 305.459,Z 395.915,A -85,B 0,C 180,E1 -16055.113,E2 -16055.113} C_VEL
LIN {X 0,Y 305.464,Z 395.935,A -85,B 0,C 180,E1 -16058.532,E2 -16058.532} C_VEL
LIN {X 0,Y 305.456,Z 395.933,A -85,B 0,C 180,E1 -16062.586,E2 -16062.586} C_VEL
LIN {X 0,Y 305.44,Z 395.901,A -85,B 0,C 180,E1 -16066.348,E2 -16066.348} C_VEL
LIN {X 0,Y 305.46,Z 395.904,A -85,B 0,C 180,E1 -16069.893,E2 -16069.893} C_VEL
LIN {X 0,Y 305.5,Z 395.921,A -85,B 0,C 180,E1 -16073.264,E2 -16073.264} C_VEL
LIN {X 0,Y 305.461,Z 395.91,A -85,B 0,C 180,E1 -16076.483,E2 -16076.483} C_VEL
LIN {X 0,Y 305.459,Z 395.919,A -85,B 0,C 180,E1 -16079.591,E2 -16079.591} C_VEL
LIN {X 0,Y 305.539,Z 396.142,A -85,B 0,C 180,E1 -16083.02,E2 -16083.02} C_VEL
LIN {X 0,Y 305.766,Z 397.099,A -85,B 0,C 180,E1 -16083.25,E2 -16083.25} C_VEL
LIN {X 0,Y 309.591,Z 403.705,A -85,B 0,C 180,E1 -16083.846,E2 -16083.846} C_VEL
LIN {X 0,Y 312.826,Z 408.448,A -85,B 0,C 180,E1 -16084.343,E2 -16084.343} C_VEL
LIN {X 0,Y 316.622,Z 413.565,A -85,B 0,C 180,E1 -16084.934,E2 -16084.934} C_VEL
LIN {X 0,Y 324.341,Z 422.831,A -85,B 0,C 180,E1 -16086.261,E2 -16086.261} C_VEL
LIN {X 0,Y 331.496,Z 430.684,A -85,B 0,C 180,E1 -16087.635,E2 -16087.635} C_VEL
LIN {X 0,Y 337.794,Z 437.165,A -85,B 0,C 180,E1 -16088.948,E2 -16088.948} C_VEL
LIN {X 0,Y 344.172,Z 443.517,A -85,B 0,C 180,E1 -16090.372,E2 -16090.372} C_VEL
LIN {X 0,Y 347.622,Z 446.663,A -85,B 0,C 180,E1 -16091.179,E2 -16091.179} C_VEL
LIN {X 0,Y 352.95,Z 451.365,A -85,B 0,C 180,E1 -16092.517,E2 -16092.517} C_VEL
LIN {X 0,Y 356.078,Z 454.184,A -85,B 0,C 180,E1 -16093.362,E2 -16093.362} C_VEL
LIN {X 0,Y 360.76,Z 458.199,A -85,B 0,C 180,E1 -16094.716,E2 -16094.716} C_VEL
LIN {X 0,Y 364.438,Z 461.147,A -85,B 0,C 180,E1 -16095.869,E2 -16095.869} C_VEL
LIN {X 0,Y 368.754,Z 464.892,A -85,B 0,C 180,E1 -16097.378,E2 -16097.378} C_VEL
LIN {X 0,Y 372.511,Z 467.383,A -85,B 0,C 180,E1 -16098.827,E2 -16098.827} C_VEL
LIN {X 0,Y 374.582,Z 468.71,A -85,B 0,C 180,E1 -16099.7,E2 -16099.7} C_VEL
LIN {X 0,Y 377.881,Z 471.893,A -85,B 0,C 180,E1 -16101.376,E2 -16101.376} C_VEL
LIN {X 0,Y 380.706,Z 473.937,A -85,B 0,C 180,E1 -16103.09,E2 -16103.09} C_VEL
LIN {X 0,Y 383.172,Z 475.284,A -85,B 0,C 180,E1 -16105.011,E2 -16105.011} C_VEL
LIN {X 0,Y 384.859,Z 475.829,A -85,B 0,C 180,E1 -16106.859,E2 -16106.859} C_VEL
LIN {X 0,Y 385.794,Z 476.43,A -85,B 0,C 180,E1 -16108.956,E2 -16108.956} C_VEL
LIN {X 0,Y 385.946,Z 476.368,A -85,B 0,C 180,E1 -16110,E2 -16110} C_VEL
LIN {X 0,Y 385.654,Z 476.305,A -85,B 0,C 180,E1 -16111.566,E2 -16111.566} C_VEL
LIN {X 0,Y 384.854,Z 475.866,A -85,B 0,C 180,E1 -16113.14,E2 -16113.14} C_VEL
LIN {X 0,Y 383.172,Z 475.295,A -85,B 0,C 180,E1 -16114.988,E2 -16114.988} C_VEL
LIN {X 0,Y 380.706,Z 473.936,A -85,B 0,C 180,E1 -16116.91,E2 -16116.91} C_VEL
LIN {X 0,Y 377.564,Z 471.656,A -85,B 0,C 180,E1 -16118.792,E2 -16118.792} C_VEL
LIN {X 0,Y 373.599,Z 467.955,A -85,B 0,C 180,E1 -16120.731,E2 -16120.731} C_VEL
LIN {X 0,Y 369.5,Z 465.449,A -85,B 0,C 180,E1 -16122.348,E2 -16122.348} C_VEL
LIN {X 0,Y 365.06,Z 461.72,A -85,B 0,C 180,E1 -16123.923,E2 -16123.923} C_VEL
LIN {X 0,Y 362.242,Z 459.277,A -85,B 0,C 180,E1 -16124.835,E2 -16124.835} C_VEL
LIN {X 0,Y 357.213,Z 455.276,A -85,B 0,C 180,E1 -16126.317,E2 -16126.317} C_VEL
LIN {X 0,Y 353.195,Z 451.538,A -85,B 0,C 180,E1 -16127.421,E2 -16127.421} C_VEL
LIN {X 0,Y 347.95,Z 447.015,A -85,B 0,C 180,E1 -16128.739,E2 -16128.739} C_VEL
LIN {X 0,Y 343.795,Z 443.143,A -85,B 0,C 180,E1 -16129.716,E2 -16129.716} C_VEL
LIN {X 0,Y 339.323,Z 438.615,A -85,B 0,C 180,E1 -16130.73,E2 -16130.73} C_VEL
LIN {X 0,Y 333.622,Z 432.865,A -85,B 0,C 180,E1 -16131.94,E2 -16131.94} C_VEL
LIN {X 0,Y 327.47,Z 426.264,A -85,B 0,C 180,E1 -16133.154,E2 -16133.154} C_VEL
LIN {X 0,Y 322.156,Z 420.098,A -85,B 0,C 180,E1 -16134.139,E2 -16134.139} C_VEL
LIN {X 0,Y 317.781,Z 414.936,A -85,B 0,C 180,E1 -16134.876,E2 -16134.876} C_VEL
LIN {X 0,Y 313.706,Z 409.766,A -85,B 0,C 180,E1 -16135.518,E2 -16135.518} C_VEL
LIN {X 0,Y 309.975,Z 404.246,A -85,B 0,C 180,E1 -16136.099,E2 -16136.099} C_VEL
LIN {X 0,Y 307.415,Z 400.131,A -85,B 0,C 180,E1 -16136.471,E2 -16136.471} C_VEL
LIN {X 0,Y 305.694,Z 396.845,A -85,B 0,C 180,E1 -16136.785,E2 -16136.785} C_VEL
LIN {X 0,Y 305.506,Z 396.025,A -85,B 0,C 180,E1 -16137.072,E2 -16137.072} C_VEL
LIN {X 0,Y 305.457,Z 395.92,A -85,B 0,C 180,E1 -16140.409,E2 -16140.409} C_VEL
LIN {X 0,Y 305.459,Z 395.904,A -85,B 0,C 180,E1 -16144.078,E2 -16144.078} C_VEL
LIN {X 0,Y 305.498,Z 395.922,A -85,B 0,C 180,E1 -16146.735,E2 -16146.735} C_VEL
LIN {X 0,Y 305.458,Z 395.905,A -85,B 0,C 180,E1 -16150.107,E2 -16150.107} C_VEL
LIN {X 0,Y 305.438,Z 395.901,A -85,B 0,C 180,E1 -16153.652,E2 -16153.652} C_VEL
LIN {X 0,Y 305.489,Z 395.929,A -85,B 0,C 180,E1 -16157.406,E2 -16157.406} C_VEL
LIN {X 0,Y 305.512,Z 395.929,A -85,B 0,C 180,E1 -16161.604,E2 -16161.604} C_VEL
LIN {X 0,Y 305.456,Z 395.916,A -85,B 0,C 180,E1 -16164.887,E2 -16164.887} C_VEL
LIN {X 0,Y 305.445,Z 395.938,A -85,B 0,C 180,E1 -16168.355,E2 -16168.355} C_VEL
LIN {X 0,Y 305.514,Z 395.914,A -85,B 0,C 180,E1 -16171.114,E2 -16171.114} C_VEL
LIN {X 0,Y 305.565,Z 395.907,A -85,B 0,C 180,E1 -16174.088,E2 -16174.088} C_VEL
LIN {X 0,Y 305.493,Z 395.92,A -85,B 0,C 180,E1 -16178.403,E2 -16178.403} C_VEL
LIN {X 0,Y 305.583,Z 395.889,A -85,B 0,C 180,E1 -16181.218,E2 -16181.218} C_VEL
LIN {X 0,Y 305.643,Z 395.911,A -85,B 0,C 180,E1 -16185.35,E2 -16185.35} C_VEL
LIN {X 0,Y 305.634,Z 395.879,A -85,B 0,C 180,E1 -16189.4,E2 -16189.4} C_VEL
LIN {X 0,Y 305.807,Z 395.875,A -85,B 0,C 180,E1 -16192.075,E2 -16192.075} C_VEL
LIN {X 0,Y 305.685,Z 395.908,A -85,B 0,C 180,E1 -16194.724,E2 -16194.724} C_VEL
LIN {X 0,Y 305.952,Z 395.84,A -85,B 0,C 180,E1 -16198.684,E2 -16198.684} C_VEL
LIN {X 0,Y 305.952,Z 395.852,A -85,B 0,C 180,E1 -16201.317,E2 -16201.317} C_VEL
LIN {X 0,Y 305.892,Z 395.865,A -85,B 0,C 180,E1 -16202.07,E2 -16202.07} C_VEL
LIN {X 0,Y 305.187,Z 395.966,A -85,B 0,C 180,E1 -16203.167,E2 -16203.167} C_VEL
LIN {X 0,Y 302.288,Z 396.329,A -85,B 0,C 180,E1 -16204.952,E2 -16204.952} C_VEL
LIN {X 0,Y 299.856,Z 396.624,A -85,B 0,C 180,E1 -16206.4,E2 -16206.4} C_VEL
LIN {X 0,Y 298.827,Z 396.74,A -85,B 0,C 180,E1 -16207.522,E2 -16207.522} C_VEL
LIN {X 0,Y 298.75,Z 396.741,A -85,B 0,C 180,E1 -16207.903,E2 -16207.903} C_VEL
LIN {X 0,Y 298.589,Z 396.762,A -85,B 0,C 180,E1 -16210.854,E2 -16210.854} C_VEL
LIN {X 0,Y 298.602,Z 396.783,A -85,B 0,C 180,E1 -16215.21,E2 -16215.21} C_VEL
LIN {X 0,Y 298.535,Z 396.766,A -85,B 0,C 180,E1 -16219.244,E2 -16219.244} C_VEL
LIN {X 0,Y 298.454,Z 396.806,A -85,B 0,C 180,E1 -16223.599,E2 -16223.599} C_VEL
LIN {X 0,Y 298.487,Z 396.775,A -85,B 0,C 180,E1 -16226.575,E2 -16226.575} C_VEL
LIN {X 0,Y 298.42,Z 396.809,A -85,B 0,C 180,E1 -16229.642,E2 -16229.642} C_VEL
LIN {X 0,Y 298.395,Z 396.801,A -85,B 0,C 180,E1 -16232.801,E2 -16232.801} C_VEL
LIN {X 0,Y 298.469,Z 396.806,A -85,B 0,C 180,E1 -16236.815,E2 -16236.815} C_VEL
LIN {X 0,Y 298.455,Z 396.804,A -85,B 0,C 180,E1 -16241.251,E2 -16241.251} C_VEL
LIN {X 0,Y 298.416,Z 396.808,A -85,B 0,C 180,E1 -16245.048,E2 -16245.048} C_VEL
LIN {X 0,Y 298.387,Z 396.788,A -85,B 0,C 180,E1 -16248.913,E2 -16248.913} C_VEL
LIN {X 0,Y 298.426,Z 396.811,A -85,B 0,C 180,E1 -16252.245,E2 -16252.245} C_VEL
LIN {X 0,Y 298.47,Z 396.944,A -85,B 0,C 180,E1 -16254.547,E2 -16254.547} C_VEL
LIN {X 0,Y 299.929,Z 403.859,A -85,B 0,C 180,E1 -16257.519,E2 -16257.519} C_VEL
LIN {X 0,Y 301.445,Z 411.492,A -85,B 0,C 180,E1 -16260.686,E2 -16260.686} C_VEL
LIN {X 0,Y 302.319,Z 417.384,A -85,B 0,C 180,E1 -16263,E2 -16263} C_VEL
LIN {X 0,Y 303.123,Z 421.025,A -85,B 0,C 180,E1 -16263.251,E2 -16263.251} C_VEL
LIN {X 0,Y 308.645,Z 447.182,A -85,B 0,C 180,E1 -16264.424,E2 -16264.424} C_VEL
LIN {X 0,Y 311.158,Z 462.24,A -85,B 0,C 180,E1 -16265.019,E2 -16265.019} C_VEL
LIN {X 0,Y 309.629,Z 522.438,A -85,B 0,C 180,E1 -16266.419,E2 -16266.419} C_VEL
LIN {X 0,Y 309.012,Z 533.15,A -85,B 0,C 180,E1 -16266.813,E2 -16266.813} C_VEL
LIN {X 0,Y 308.227,Z 542.272,A -85,B 0,C 180,E1 -16267.283,E2 -16267.283} C_VEL
LIN {X 0,Y 307.142,Z 552.626,A -85,B 0,C 180,E1 -16267.995,E2 -16267.995} C_VEL
LIN {X 0,Y 306.094,Z 561.772,A -85,B 0,C 180,E1 -16268.801,E2 -16268.801} C_VEL
LIN {X 0,Y 304.801,Z 570.77,A -85,B 0,C 180,E1 -16269.766,E2 -16269.766} C_VEL
LIN {X 0,Y 303.435,Z 579.494,A -85,B 0,C 180,E1 -16270.904,E2 -16270.904} C_VEL
LIN {X 0,Y 302.288,Z 586.916,A -85,B 0,C 180,E1 -16272.059,E2 -16272.059} C_VEL
LIN {X 0,Y 301.157,Z 594.392,A -85,B 0,C 180,E1 -16273.443,E2 -16273.443} C_VEL
LIN {X 0,Y 299.918,Z 601.705,A -85,B 0,C 180,E1 -16275.063,E2 -16275.063} C_VEL
LIN {X 0,Y 298.809,Z 608.015,A -85,B 0,C 180,E1 -16276.744,E2 -16276.744} C_VEL
LIN {X 0,Y 297.955,Z 613.288,A -85,B 0,C 180,E1 -16278.435,E2 -16278.435} C_VEL
LIN {X 0,Y 297.245,Z 618.384,A -85,B 0,C 180,E1 -16280.474,E2 -16280.474} C_VEL
LIN {X 0,Y 296.791,Z 622.35,A -85,B 0,C 180,E1 -16282.517,E2 -16282.517} C_VEL
LIN {X 0,Y 296.554,Z 625.287,A -85,B 0,C 180,E1 -16284.561,E2 -16284.561} C_VEL
LIN {X 0,Y 296.5,Z 626.788,A -85,B 0,C 180,E1 -16285.923,E2 -16285.923} C_VEL
LIN {X 0,Y 296.529,Z 627.719,A -85,B 0,C 180,E1 -16287.283,E2 -16287.283} C_VEL
LIN {X 0,Y 296.507,Z 628.593,A -85,B 0,C 180,E1 -16290,E2 -16290} C_VEL
LIN {X 0,Y 296.528,Z 627.718,A -85,B 0,C 180,E1 -16292.717,E2 -16292.717} C_VEL
LIN {X 0,Y 296.494,Z 626.788,A -85,B 0,C 180,E1 -16294.078,E2 -16294.078} C_VEL
LIN {X 0,Y 296.665,Z 623.438,A -85,B 0,C 180,E1 -16296.803,E2 -16296.803} C_VEL
LIN {X 0,Y 297.062,Z 619.81,A -85,B 0,C 180,E1 -16298.846,E2 -16298.846} C_VEL
LIN {X 0,Y 297.7,Z 615.077,A -85,B 0,C 180,E1 -16300.887,E2 -16300.887} C_VEL
LIN {X 0,Y 298.423,Z 610.196,A -85,B 0,C 180,E1 -16302.583,E2 -16302.583} C_VEL
LIN {X 0,Y 299.45,Z 604.325,A -85,B 0,C 180,E1 -16304.267,E2 -16304.267} C_VEL
LIN {X 0,Y 300.377,Z 598.832,A -85,B 0,C 180,E1 -16305.609,E2 -16305.609} C_VEL
LIN {X 0,Y 301.708,Z 590.806,A -85,B 0,C 180,E1 -16307.241,E2 -16307.241} C_VEL
LIN {X 0,Y 302.961,Z 582.785,A -85,B 0,C 180,E1 -16308.601,E2 -16308.601} C_VEL
LIN {X 0,Y 304.227,Z 574.702,A -85,B 0,C 180,E1 -16309.746,E2 -16309.746} C_VEL
LIN {X 0,Y 305.608,Z 564.942,A -85,B 0,C 180,E1 -16310.883,E2 -16310.883} C_VEL
LIN {X 0,Y 306.76,Z 556.555,A -85,B 0,C 180,E1 -16311.681,E2 -16311.681} C_VEL
LIN {X 0,Y 307.864,Z 546.047,A -85,B 0,C 180,E1 -16312.481,E2 -16312.481} C_VEL
LIN {X 0,Y 308.814,Z 535.716,A -85,B 0,C 180,E1 -16313.071,E2 -16313.071} C_VEL
LIN {X 0,Y 309.573,Z 524.997,A -85,B 0,C 180,E1 -16313.498,E2 -16313.498} C_VEL
LIN {X 0,Y 310.196,Z 501.202,A -85,B 0,C 180,E1 -16314.093,E2 -16314.093} C_VEL
LIN {X 0,Y 311.021,Z 460.91,A -85,B 0,C 180,E1 -16315.026,E2 -16315.026} C_VEL
LIN {X 0,Y 306.927,Z 438.364,A -85,B 0,C 180,E1 -16315.953,E2 -16315.953} C_VEL
LIN {X 0,Y 302.383,Z 417.958,A -85,B 0,C 180,E1 -16316.92,E2 -16316.92} C_VEL
LIN {X 0,Y 302.283,Z 416.869,A -85,B 0,C 180,E1 -16317.148,E2 -16317.148} C_VEL
LIN {X 0,Y 301.018,Z 409.206,A -85,B 0,C 180,E1 -16320.246,E2 -16320.246} C_VEL
LIN {X 0,Y 299.22,Z 400.474,A -85,B 0,C 180,E1 -16323.906,E2 -16323.906} C_VEL
LIN {X 0,Y 298.458,Z 396.866,A -85,B 0,C 180,E1 -16325.56,E2 -16325.56} C_VEL
LIN {X 0,Y 298.411,Z 396.793,A -85,B 0,C 180,E1 -16329.486,E2 -16329.486} C_VEL
LIN {X 0,Y 298.428,Z 396.81,A -85,B 0,C 180,E1 -16333.108,E2 -16333.108} C_VEL
LIN {X 0,Y 298.47,Z 396.804,A -85,B 0,C 180,E1 -16336.932,E2 -16336.932} C_VEL
LIN {X 0,Y 298.442,Z 396.8,A -85,B 0,C 180,E1 -16340.997,E2 -16340.997} C_VEL
LIN {X 0,Y 298.436,Z 396.805,A -85,B 0,C 180,E1 -16343.932,E2 -16343.932} C_VEL
LIN {X 0,Y 298.4,Z 396.807,A -85,B 0,C 180,E1 -16347.982,E2 -16347.982} C_VEL
LIN {X 0,Y 298.465,Z 396.787,A -85,B 0,C 180,E1 -16351.904,E2 -16351.904} C_VEL
LIN {X 0,Y 298.486,Z 396.79,A -85,B 0,C 180,E1 -16354.923,E2 -16354.923} C_VEL
LIN {X 0,Y 298.45,Z 396.793,A -85,B 0,C 180,E1 -16359.315,E2 -16359.315} C_VEL
LIN {X 0,Y 298.538,Z 396.765,A -85,B 0,C 180,E1 -16362.179,E2 -16362.179} C_VEL
LIN {X 0,Y 298.593,Z 396.785,A -85,B 0,C 180,E1 -16364.994,E2 -16364.994} C_VEL
LIN {X 0,Y 298.593,Z 396.761,A -85,B 0,C 180,E1 -16369.146,E2 -16369.146} C_VEL
LIN {X 0,Y 298.759,Z 396.737,A -85,B 0,C 180,E1 -16371.885,E2 -16371.885} C_VEL
LIN {X 0,Y 298.659,Z 396.78,A -85,B 0,C 180,E1 -16374.598,E2 -16374.598} C_VEL
LIN {X 0,Y 298.923,Z 396.727,A -85,B 0,C 180,E1 -16378.652,E2 -16378.652} C_VEL
LIN {X 0,Y 298.921,Z 396.715,A -85,B 0,C 180,E1 -16381.346,E2 -16381.346} C_VEL
LIN {X 0,Y 298.796,Z 396.761,A -85,B 0,C 180,E1 -16386.753,E2 -16386.753} C_VEL
LIN {X 0,Y 298.679,Z 396.745,A -85,B 0,C 180,E1 -16389.48,E2 -16389.48} C_VEL
LIN {X 0,Y 298.551,Z 396.792,A -85,B 0,C 180,E1 -16393.615,E2 -16393.615} C_VEL
LIN {X 0,Y 298.547,Z 396.79,A -85,B 0,C 180,E1 -16396.408,E2 -16396.408} C_VEL
LIN {X 0,Y 298.509,Z 396.77,A -85,B 0,C 180,E1 -16399.654,E2 -16399.654} C_VEL
LIN {X 0,Y 298.455,Z 396.81,A -85,B 0,C 180,E1 -16403.597,E2 -16403.597} C_VEL
LIN {X 0,Y 298.484,Z 396.782,A -85,B 0,C 180,E1 -16406.574,E2 -16406.574} C_VEL
LIN {X 0,Y 298.413,Z 396.806,A -85,B 0,C 180,E1 -16409.641,E2 -16409.641} C_VEL
LIN {X 0,Y 298.391,Z 396.809,A -85,B 0,C 180,E1 -16412.8,E2 -16412.8} C_VEL
LIN {X 0,Y 298.461,Z 396.804,A -85,B 0,C 180,E1 -16416.812,E2 -16416.812} C_VEL
LIN {X 0,Y 298.384,Z 396.8,A -85,B 0,C 180,E1 -16421.087,E2 -16421.087} C_VEL
LIN {X 0,Y 298.385,Z 396.803,A -85,B 0,C 180,E1 -16425.041,E2 -16425.041} C_VEL
LIN {X 0,Y 298.388,Z 396.768,A -85,B 0,C 180,E1 -16428.911,E2 -16428.911} C_VEL
LIN {X 0,Y 298.445,Z 396.811,A -85,B 0,C 180,E1 -16432.246,E2 -16432.246} C_VEL
LIN {X 0,Y 298.405,Z 396.781,A -85,B 0,C 180,E1 -16435.581,E2 -16435.581} C_VEL
LIN {X 0,Y 298.392,Z 396.812,A -85,B 0,C 180,E1 -16438.791,E2 -16438.791} C_VEL
LIN {X 0,Y 298.483,Z 396.97,A -85,B 0,C 180,E1 -16442.324,E2 -16442.324} C_VEL
LIN {X 0,Y 298.791,Z 398.117,A -85,B 0,C 180,E1 -16442.596,E2 -16442.596} C_VEL
LIN {X 0,Y 303.598,Z 406.919,A -85,B 0,C 180,E1 -16443.316,E2 -16443.316} C_VEL
LIN {X 0,Y 310.878,Z 417.179,A -85,B 0,C 180,E1 -16444.347,E2 -16444.347} C_VEL
LIN {X 0,Y 318.558,Z 426.107,A -85,B 0,C 180,E1 -16445.538,E2 -16445.538} C_VEL
LIN {X 0,Y 326.455,Z 434.866,A -85,B 0,C 180,E1 -16446.937,E2 -16446.937} C_VEL
LIN {X 0,Y 334.629,Z 443.092,A -85,B 0,C 180,E1 -16448.546,E2 -16448.546} C_VEL
LIN {X 0,Y 341.793,Z 450.024,A -85,B 0,C 180,E1 -16450.101,E2 -16450.101} C_VEL
LIN {X 0,Y 348.765,Z 456.353,A -85,B 0,C 180,E1 -16451.751,E2 -16451.751} C_VEL
LIN {X 0,Y 353.426,Z 460.23,A -85,B 0,C 180,E1 -16452.937,E2 -16452.937} C_VEL
LIN {X 0,Y 358.648,Z 464.712,A -85,B 0,C 180,E1 -16454.399,E2 -16454.399} C_VEL
LIN {X 0,Y 362.731,Z 467.893,A -85,B 0,C 180,E1 -16455.638,E2 -16455.638} C_VEL
LIN {X 0,Y 367.468,Z 471.881,A -85,B 0,C 180,E1 -16457.261,E2 -16457.261} C_VEL
LIN {X 0,Y 371.705,Z 474.558,A -85,B 0,C 180,E1 -16458.88,E2 -16458.88} C_VEL
LIN {X 0,Y 373.719,Z 476.108,A -85,B 0,C 180,E1 -16459.744,E2 -16459.744} C_VEL
LIN {X 0,Y 377.193,Z 479.236,A -85,B 0,C 180,E1 -16461.505,E2 -16461.505} C_VEL
LIN {X 0,Y 380.083,Z 481.158,A -85,B 0,C 180,E1 -16463.274,E2 -16463.274} C_VEL
LIN {X 0,Y 382.595,Z 482.444,A -85,B 0,C 180,E1 -16465.263,E2 -16465.263} C_VEL
LIN {X 0,Y 384.297,Z 483.053,A -85,B 0,C 180,E1 -16467.367,E2 -16467.367} C_VEL
LIN {X 0,Y 384.932,Z 483.473,A -85,B 0,C 180,E1 -16468.954,E2 -16468.954} C_VEL
LIN {X 0,Y 385.081,Z 483.415,A -85,B 0,C 180,E1 -16470,E2 -16470} C_VEL
LIN {X 0,Y 384.785,Z 483.353,A -85,B 0,C 180,E1 -16471.57,E2 -16471.57} C_VEL
LIN {X 0,Y 383.979,Z 482.891,A -85,B 0,C 180,E1 -16473.147,E2 -16473.147} C_VEL
LIN {X 0,Y 382.281,Z 482.341,A -85,B 0,C 180,E1 -16475,E2 -16475} C_VEL
LIN {X 0,Y 379.792,Z 480.989,A -85,B 0,C 180,E1 -16476.927,E2 -16476.927} C_VEL
LIN {X 0,Y 376.551,Z 478.743,A -85,B 0,C 180,E1 -16478.839,E2 -16478.839} C_VEL
LIN {X 0,Y 372.964,Z 475.382,A -85,B 0,C 180,E1 -16480.595,E2 -16480.595} C_VEL
LIN {X 0,Y 368.235,Z 472.433,A -85,B 0,C 180,E1 -16482.456,E2 -16482.456} C_VEL
LIN {X 0,Y 363.701,Z 468.782,A -85,B 0,C 180,E1 -16484.037,E2 -16484.037} C_VEL
LIN {X 0,Y 360.203,Z 465.834,A -85,B 0,C 180,E1 -16485.144,E2 -16485.144} C_VEL
LIN {X 0,Y 354.989,Z 461.728,A -85,B 0,C 180,E1 -16486.632,E2 -16486.632} C_VEL
LIN {X 0,Y 350.414,Z 457.623,A -85,B 0,C 180,E1 -16487.848,E2 -16487.848} C_VEL
LIN {X 0,Y 344.835,Z 452.804,A -85,B 0,C 180,E1 -16489.203,E2 -16489.203} C_VEL
LIN {X 0,Y 337.919,Z 446.423,A -85,B 0,C 180,E1 -16490.748,E2 -16490.748} C_VEL
LIN {X 0,Y 330.378,Z 438.826,A -85,B 0,C 180,E1 -16492.313,E2 -16492.313} C_VEL
LIN {X 0,Y 323.584,Z 431.635,A -85,B 0,C 180,E1 -16493.601,E2 -16493.601} C_VEL
LIN {X 0,Y 315.997,Z 423.259,A -85,B 0,C 180,E1 -16494.874,E2 -16494.874} C_VEL
LIN {X 0,Y 309.289,Z 415.037,A -85,B 0,C 180,E1 -16495.885,E2 -16495.885} C_VEL
LIN {X 0,Y 302.851,Z 405.731,A -85,B 0,C 180,E1 -16496.786,E2 -16496.786} C_VEL
LIN {X 0,Y 298.713,Z 397.934,A -85,B 0,C 180,E1 -16497.428,E2 -16497.428} C_VEL
LIN {X 0,Y 298.489,Z 396.903,A -85,B 0,C 180,E1 -16497.726,E2 -16497.726} C_VEL
LIN {X 0,Y 298.391,Z 396.817,A -85,B 0,C 180,E1 -16502.017,E2 -16502.017} C_VEL
LIN {X 0,Y 298.428,Z 396.789,A -85,B 0,C 180,E1 -16506.067,E2 -16506.067} C_VEL
LIN {X 0,Y 298.413,Z 396.795,A -85,B 0,C 180,E1 -16509.484,E2 -16509.484} C_VEL
LIN {X 0,Y 298.392,Z 396.768,A -85,B 0,C 180,E1 -16513.103,E2 -16513.103} C_VEL
LIN {X 0,Y 298.426,Z 396.812,A -85,B 0,C 180,E1 -16516.926,E2 -16516.926} C_VEL
LIN {X 0,Y 298.425,Z 396.808,A -85,B 0,C 180,E1 -16521,E2 -16521} C_VEL
LIN {X 0,Y 298.427,Z 396.802,A -85,B 0,C 180,E1 -16523.932,E2 -16523.932} C_VEL
LIN {X 0,Y 298.389,Z 396.814,A -85,B 0,C 180,E1 -16527.984,E2 -16527.984} C_VEL
LIN {X 0,Y 298.457,Z 396.784,A -85,B 0,C 180,E1 -16531.905,E2 -16531.905} C_VEL
LIN {X 0,Y 298.479,Z 396.798,A -85,B 0,C 180,E1 -16534.924,E2 -16534.924} C_VEL
LIN {X 0,Y 298.443,Z 396.789,A -85,B 0,C 180,E1 -16539.316,E2 -16539.316} C_VEL
LIN {X 0,Y 298.531,Z 396.775,A -85,B 0,C 180,E1 -16542.18,E2 -16542.18} C_VEL
LIN {X 0,Y 298.588,Z 396.791,A -85,B 0,C 180,E1 -16544.995,E2 -16544.995} C_VEL
LIN {X 0,Y 298.589,Z 396.757,A -85,B 0,C 180,E1 -16549.147,E2 -16549.147} C_VEL
LIN {X 0,Y 298.753,Z 396.752,A -85,B 0,C 180,E1 -16551.887,E2 -16551.887} C_VEL
LIN {X 0,Y 298.656,Z 396.784,A -85,B 0,C 180,E1 -16554.6,E2 -16554.6} C_VEL
LIN {X 0,Y 298.919,Z 396.715,A -85,B 0,C 180,E1 -16558.654,E2 -16558.654} C_VEL
LIN {X 0,Y 298.919,Z 396.727,A -85,B 0,C 180,E1 -16561.348,E2 -16561.348} C_VEL
LIN {X 0,Y 298.794,Z 396.753,A -85,B 0,C 180,E1 -16566.755,E2 -16566.755} C_VEL
LIN {X 0,Y 298.75,Z 396.741,A -85,B 0,C 180,E1 -16567.903,E2 -16567.903} C_VEL
LIN {X 0,Y 298.07,Z 396.82,A -85,B 0,C 180,E1 -16569.026,E2 -16569.026} C_VEL
LIN {X 0,Y 295.109,Z 397.195,A -85,B 0,C 180,E1 -16570.852,E2 -16570.852} C_VEL
LIN {X 0,Y 292.613,Z 397.524,A -85,B 0,C 180,E1 -16572.334,E2 -16572.334} C_VEL
LIN {X 0,Y 291.578,Z 397.66,A -85,B 0,C 180,E1 -16573.485,E2 -16573.485} C_VEL
LIN {X 0,Y 291.513,Z 397.669,A -85,B 0,C 180,E1 -16573.875,E2 -16573.875} C_VEL
LIN {X 0,Y 291.483,Z 397.655,A -85,B 0,C 180,E1 -16576.819,E2 -16576.819} C_VEL
LIN {X 0,Y 291.447,Z 397.655,A -85,B 0,C 180,E1 -16579.876,E2 -16579.876} C_VEL
LIN {X 0,Y 291.397,Z 397.678,A -85,B 0,C 180,E1 -16584.206,E2 -16584.206} C_VEL
LIN {X 0,Y 291.42,Z 397.656,A -85,B 0,C 180,E1 -16587.273,E2 -16587.273} C_VEL
LIN {X 0,Y 291.338,Z 397.696,A -85,B 0,C 180,E1 -16590.438,E2 -16590.438} C_VEL
LIN {X 0,Y 291.344,Z 397.672,A -85,B 0,C 180,E1 -16593.699,E2 -16593.699} C_VEL
LIN {X 0,Y 291.404,Z 397.686,A -85,B 0,C 180,E1 -16597.263,E2 -16597.263} C_VEL
LIN {X 0,Y 291.405,Z 397.676,A -85,B 0,C 180,E1 -16600.631,E2 -16600.631} C_VEL
LIN {X 0,Y 291.352,Z 397.684,A -85,B 0,C 180,E1 -16604.391,E2 -16604.391} C_VEL
LIN {X 0,Y 291.331,Z 397.67,A -85,B 0,C 180,E1 -16608.404,E2 -16608.404} C_VEL
LIN {X 0,Y 291.364,Z 397.681,A -85,B 0,C 180,E1 -16611.161,E2 -16611.161} C_VEL
LIN {X 0,Y 291.426,Z 397.807,A -85,B 0,C 180,E1 -16613.998,E2 -16613.998} C_VEL
LIN {X 0,Y 293.427,Z 407.297,A -85,B 0,C 180,E1 -16618.203,E2 -16618.203} C_VEL
LIN {X 0,Y 294.571,Z 413.225,A -85,B 0,C 180,E1 -16620.72,E2 -16620.72} C_VEL
LIN {X 0,Y 295.247,Z 417.202,A -85,B 0,C 180,E1 -16622.304,E2 -16622.304} C_VEL
LIN {X 0,Y 296.619,Z 421.635,A -85,B 0,C 180,E1 -16622.637,E2 -16622.637} C_VEL
LIN {X 0,Y 301.517,Z 444.658,A -85,B 0,C 180,E1 -16623.714,E2 -16623.714} C_VEL
LIN {X 0,Y 304.732,Z 463.094,A -85,B 0,C 180,E1 -16624.481,E2 -16624.481} C_VEL
LIN {X 0,Y 303.13,Z 522.249,A -85,B 0,C 180,E1 -16625.882,E2 -16625.882} C_VEL
LIN {X 0,Y 302.51,Z 532.956,A -85,B 0,C 180,E1 -16626.284,E2 -16626.284} C_VEL
LIN {X 0,Y 301.696,Z 542.078,A -85,B 0,C 180,E1 -16626.762,E2 -16626.762} C_VEL
LIN {X 0,Y 300.567,Z 552.431,A -85,B 0,C 180,E1 -16627.488,E2 -16627.488} C_VEL
LIN {X 0,Y 299.489,Z 561.577,A -85,B 0,C 180,E1 -16628.31,E2 -16628.31} C_VEL
LIN {X 0,Y 298.148,Z 570.575,A -85,B 0,C 180,E1 -16629.294,E2 -16629.294} C_VEL
LIN {X 0,Y 296.721,Z 579.299,A -85,B 0,C 180,E1 -16630.455,E2 -16630.455} C_VEL
LIN {X 0,Y 295.507,Z 586.72,A -85,B 0,C 180,E1 -16631.632,E2 -16631.632} C_VEL
LIN {X 0,Y 294.099,Z 595.519,A -85,B 0,C 180,E1 -16633.337,E2 -16633.337} C_VEL
LIN {X 0,Y 293.029,Z 601.509,A -85,B 0,C 180,E1 -16634.704,E2 -16634.704} C_VEL
LIN {X 0,Y 291.886,Z 607.819,A -85,B 0,C 180,E1 -16636.423,E2 -16636.423} C_VEL
LIN {X 0,Y 290.965,Z 613.092,A -85,B 0,C 180,E1 -16638.153,E2 -16638.153} C_VEL
LIN {X 0,Y 290.201,Z 618.188,A -85,B 0,C 180,E1 -16640.24,E2 -16640.24} C_VEL
LIN {X 0,Y 289.722,Z 622.154,A -85,B 0,C 180,E1 -16642.333,E2 -16642.333} C_VEL
LIN {X 0,Y 289.479,Z 625.182,A -85,B 0,C 180,E1 -16644.51,E2 -16644.51} C_VEL
LIN {X 0,Y 289.405,Z 626.593,A -85,B 0,C 180,E1 -16645.823,E2 -16645.823} C_VEL
LIN {X 0,Y 289.408,Z 628.119,A -85,B 0,C 180,E1 -16648.609,E2 -16648.609} C_VEL
LIN {X 0,Y 289.425,Z 628.399,A -85,B 0,C 180,E1 -16650,E2 -16650} C_VEL
LIN {X 0,Y 289.431,Z 627.523,A -85,B 0,C 180,E1 -16652.784,E2 -16652.784} C_VEL
LIN {X 0,Y 289.399,Z 626.592,A -85,B 0,C 180,E1 -16654.178,E2 -16654.178} C_VEL
LIN {X 0,Y 289.594,Z 623.242,A -85,B 0,C 180,E1 -16656.97,E2 -16656.97} C_VEL
LIN {X 0,Y 290.029,Z 619.615,A -85,B 0,C 180,E1 -16659.063,E2 -16659.063} C_VEL
LIN {X 0,Y 290.708,Z 614.882,A -85,B 0,C 180,E1 -16661.152,E2 -16661.152} C_VEL
LIN {X 0,Y 291.443,Z 610,A -85,B 0,C 180,E1 -16662.889,E2 -16662.889} C_VEL
LIN {X 0,Y 292.557,Z 604.129,A -85,B 0,C 180,E1 -16664.61,E2 -16664.61} C_VEL
LIN {X 0,Y 293.52,Z 598.636,A -85,B 0,C 180,E1 -16665.983,E2 -16665.983} C_VEL
LIN {X 0,Y 294.783,Z 591.378,A -85,B 0,C 180,E1 -16667.511,E2 -16667.511} C_VEL
LIN {X 0,Y 296.2,Z 582.589,A -85,B 0,C 180,E1 -16669.041,E2 -16669.041} C_VEL
LIN {X 0,Y 297.54,Z 574.507,A -85,B 0,C 180,E1 -16670.209,E2 -16670.209} C_VEL
LIN {X 0,Y 298.998,Z 564.747,A -85,B 0,C 180,E1 -16671.366,E2 -16671.366} C_VEL
LIN {X 0,Y 300.162,Z 556.359,A -85,B 0,C 180,E1 -16672.182,E2 -16672.182} C_VEL
LIN {X 0,Y 301.302,Z 545.852,A -85,B 0,C 180,E1 -16672.998,E2 -16672.998} C_VEL
LIN {X 0,Y 302.303,Z 535.521,A -85,B 0,C 180,E1 -16673.597,E2 -16673.597} C_VEL
LIN {X 0,Y 303.082,Z 524.802,A -85,B 0,C 180,E1 -16674.032,E2 -16674.032} C_VEL
LIN {X 0,Y 303.7,Z 502.02,A -85,B 0,C 180,E1 -16674.617,E2 -16674.617} C_VEL
LIN {X 0,Y 304.577,Z 461.875,A -85,B 0,C 180,E1 -16675.564,E2 -16675.564} C_VEL
LIN {X 0,Y 300.502,Z 439.234,A -85,B 0,C 180,E1 -16676.523,E2 -16676.523} C_VEL
LIN {X 0,Y 296.196,Z 420.184,A -85,B 0,C 180,E1 -16677.443,E2 -16677.443} C_VEL
LIN {X 0,Y 295.247,Z 417.194,A -85,B 0,C 180,E1 -16677.696,E2 -16677.696} C_VEL
LIN {X 0,Y 293.951,Z 410.111,A -85,B 0,C 180,E1 -16680.602,E2 -16680.602} C_VEL
LIN {X 0,Y 292.248,Z 401.587,A -85,B 0,C 180,E1 -16684.284,E2 -16684.284} C_VEL
LIN {X 0,Y 291.429,Z 397.769,A -85,B 0,C 180,E1 -16686.002,E2 -16686.002} C_VEL
LIN {X 0,Y 291.39,Z 397.667,A -85,B 0,C 180,E1 -16689.483,E2 -16689.483} C_VEL
LIN {X 0,Y 291.35,Z 397.694,A -85,B 0,C 180,E1 -16693.641,E2 -16693.641} C_VEL
LIN {X 0,Y 291.402,Z 397.687,A -85,B 0,C 180,E1 -16697.522,E2 -16697.522} C_VEL
LIN {X 0,Y 291.39,Z 397.679,A -85,B 0,C 180,E1 -16701.163,E2 -16701.163} C_VEL
LIN {X 0,Y 291.388,Z 397.677,A -85,B 0,C 180,E1 -16704.629,E2 -16704.629} C_VEL
LIN {X 0,Y 291.377,Z 397.681,A -85,B 0,C 180,E1 -16707.951,E2 -16707.951} C_VEL
LIN {X 0,Y 291.384,Z 397.679,A -85,B 0,C 180,E1 -16711.158,E2 -16711.158} C_VEL
LIN {X 0,Y 291.417,Z 397.66,A -85,B 0,C 180,E1 -16714.271,E2 -16714.271} C_VEL
LIN {X 0,Y 291.382,Z 397.687,A -85,B 0,C 180,E1 -16717.299,E2 -16717.299} C_VEL
LIN {X 0,Y 291.459,Z 397.652,A -85,B 0,C 180,E1 -16720.269,E2 -16720.269} C_VEL
LIN {X 0,Y 291.556,Z 397.661,A -85,B 0,C 180,E1 -16724.623,E2 -16724.623} C_VEL
LIN {X 0,Y 291.536,Z 397.644,A -85,B 0,C 180,E1 -16728.88,E2 -16728.88} C_VEL
LIN {X 0,Y 291.71,Z 397.611,A -85,B 0,C 180,E1 -16731.688,E2 -16731.688} C_VEL
LIN {X 0,Y 291.63,Z 397.656,A -85,B 0,C 180,E1 -16734.468,E2 -16734.468} C_VEL
LIN {X 0,Y 291.889,Z 397.602,A -85,B 0,C 180,E1 -16738.62,E2 -16738.62} C_VEL
LIN {X 0,Y 291.887,Z 397.59,A -85,B 0,C 180,E1 -16741.379,E2 -16741.379} C_VEL
LIN {X 0,Y 291.745,Z 397.639,A -85,B 0,C 180,E1 -16746.917,E2 -16746.917} C_VEL
LIN {X 0,Y 291.628,Z 397.621,A -85,B 0,C 180,E1 -16749.711,E2 -16749.711} C_VEL
LIN {X 0,Y 291.521,Z 397.672,A -85,B 0,C 180,E1 -16753.949,E2 -16753.949} C_VEL
LIN {X 0,Y 291.485,Z 397.666,A -85,B 0,C 180,E1 -16756.817,E2 -16756.817} C_VEL
LIN {X 0,Y 291.449,Z 397.65,A -85,B 0,C 180,E1 -16759.874,E2 -16759.874} C_VEL
LIN {X 0,Y 291.398,Z 397.685,A -85,B 0,C 180,E1 -16764.205,E2 -16764.205} C_VEL
LIN {X 0,Y 291.417,Z 397.658,A -85,B 0,C 180,E1 -16767.271,E2 -16767.271} C_VEL
LIN {X 0,Y 291.331,Z 397.694,A -85,B 0,C 180,E1 -16770.437,E2 -16770.437} C_VEL
LIN {X 0,Y 291.341,Z 397.675,A -85,B 0,C 180,E1 -16773.698,E2 -16773.698} C_VEL
LIN {X 0,Y 291.391,Z 397.688,A -85,B 0,C 180,E1 -16777.258,E2 -16777.258} C_VEL
LIN {X 0,Y 291.331,Z 397.678,A -85,B 0,C 180,E1 -16780.642,E2 -16780.642} C_VEL
LIN {X 0,Y 291.312,Z 397.695,A -85,B 0,C 180,E1 -16784.397,E2 -16784.397} C_VEL
LIN {X 0,Y 291.326,Z 397.642,A -85,B 0,C 180,E1 -16788.403,E2 -16788.403} C_VEL
LIN {X 0,Y 291.378,Z 397.685,A -85,B 0,C 180,E1 -16791.162,E2 -16791.162} C_VEL
LIN {X 0,Y 291.383,Z 397.657,A -85,B 0,C 180,E1 -16794.629,E2 -16794.629} C_VEL
LIN {X 0,Y 291.37,Z 397.691,A -85,B 0,C 180,E1 -16797.95,E2 -16797.95} C_VEL
LIN {X 0,Y 291.428,Z 397.83,A -85,B 0,C 180,E1 -16801.615,E2 -16801.615} C_VEL
LIN {X 0,Y 291.705,Z 398.896,A -85,B 0,C 180,E1 -16801.889,E2 -16801.889} C_VEL
LIN {X 0,Y 298.168,Z 410.941,A -85,B 0,C 180,E1 -16802.893,E2 -16802.893} C_VEL
LIN {X 0,Y 305.817,Z 421.652,A -85,B 0,C 180,E1 -16803.928,E2 -16803.928} C_VEL
LIN {X 0,Y 312.91,Z 429.776,A -85,B 0,C 180,E1 -16804.929,E2 -16804.929} C_VEL
LIN {X 0,Y 319.07,Z 436.375,A -85,B 0,C 180,E1 -16805.89,E2 -16805.89} C_VEL
LIN {X 0,Y 324.366,Z 442.049,A -85,B 0,C 180,E1 -16806.821,E2 -16806.821} C_VEL
LIN {X 0,Y 331.283,Z 448.916,A -85,B 0,C 180,E1 -16808.14,E2 -16808.14} C_VEL
LIN {X 0,Y 339.136,Z 456.324,A -85,B 0,C 180,E1 -16809.779,E2 -16809.779} C_VEL
LIN {X 0,Y 346.398,Z 462.792,A -85,B 0,C 180,E1 -16811.454,E2 -16811.454} C_VEL
LIN {X 0,Y 350.972,Z 466.555,A -85,B 0,C 180,E1 -16812.589,E2 -16812.589} C_VEL
LIN {X 0,Y 356.403,Z 471.133,A -85,B 0,C 180,E1 -16814.062,E2 -16814.062} C_VEL
LIN {X 0,Y 360.801,Z 474.48,A -85,B 0,C 180,E1 -16815.365,E2 -16815.365} C_VEL
LIN {X 0,Y 365.505,Z 478.385,A -85,B 0,C 180,E1 -16816.91,E2 -16816.91} C_VEL
LIN {X 0,Y 369.816,Z 481.137,A -85,B 0,C 180,E1 -16818.498,E2 -16818.498} C_VEL
LIN {X 0,Y 372.05,Z 482.689,A -85,B 0,C 180,E1 -16819.424,E2 -16819.424} C_VEL
LIN {X 0,Y 375.7,Z 485.918,A -85,B 0,C 180,E1 -16821.197,E2 -16821.197} C_VEL
LIN {X 0,Y 378.87,Z 488.049,A -85,B 0,C 180,E1 -16823.056,E2 -16823.056} C_VEL
LIN {X 0,Y 381.391,Z 489.376,A -85,B 0,C 180,E1 -16824.988,E2 -16824.988} C_VEL
LIN {X 0,Y 383.299,Z 489.998,A -85,B 0,C 180,E1 -16827.103,E2 -16827.103} C_VEL
LIN {X 0,Y 384.07,Z 490.52,A -85,B 0,C 180,E1 -16828.951,E2 -16828.951} C_VEL
LIN {X 0,Y 384.216,Z 490.461,A -85,B 0,C 180,E1 -16830,E2 -16830} C_VEL
LIN {X 0,Y 383.918,Z 490.385,A -85,B 0,C 180,E1 -16831.573,E2 -16831.573} C_VEL
LIN {X 0,Y 383.105,Z 489.911,A -85,B 0,C 180,E1 -16833.154,E2 -16833.154} C_VEL
LIN {X 0,Y 381.391,Z 489.388,A -85,B 0,C 180,E1 -16835.012,E2 -16835.012} C_VEL
LIN {X 0,Y 378.869,Z 488.051,A -85,B 0,C 180,E1 -16836.944,E2 -16836.944} C_VEL
LIN {X 0,Y 375.589,Z 485.835,A -85,B 0,C 180,E1 -16838.862,E2 -16838.862} C_VEL
LIN {X 0,Y 371.927,Z 482.577,A -85,B 0,C 180,E1 -16840.631,E2 -16840.631} C_VEL
LIN {X 0,Y 368.455,Z 480.349,A -85,B 0,C 180,E1 -16842.021,E2 -16842.021} C_VEL
LIN {X 0,Y 364.155,Z 477.317,A -85,B 0,C 180,E1 -16843.549,E2 -16843.549} C_VEL
LIN {X 0,Y 358.105,Z 472.347,A -85,B 0,C 180,E1 -16845.455,E2 -16845.455} C_VEL
LIN {X 0,Y 352.564,Z 467.988,A -85,B 0,C 180,E1 -16846.996,E2 -16846.996} C_VEL
LIN {X 0,Y 347.91,Z 463.98,A -85,B 0,C 180,E1 -16848.181,E2 -16848.181} C_VEL
LIN {X 0,Y 342.167,Z 459.076,A -85,B 0,C 180,E1 -16849.534,E2 -16849.534} C_VEL
LIN {X 0,Y 334.76,Z 452.337,A -85,B 0,C 180,E1 -16851.146,E2 -16851.146} C_VEL
LIN {X 0,Y 326.867,Z 444.58,A -85,B 0,C 180,E1 -16852.716,E2 -16852.716} C_VEL
LIN {X 0,Y 320.365,Z 437.92,A -85,B 0,C 180,E1 -16853.882,E2 -16853.882} C_VEL
LIN {X 0,Y 312.443,Z 429.324,A -85,B 0,C 180,E1 -16855.14,E2 -16855.14} C_VEL
LIN {X 0,Y 304.745,Z 420.25,A -85,B 0,C 180,E1 -16856.221,E2 -16856.221} C_VEL
LIN {X 0,Y 297.626,Z 410.061,A -85,B 0,C 180,E1 -16857.184,E2 -16857.184} C_VEL
LIN {X 0,Y 291.628,Z 398.697,A -85,B 0,C 180,E1 -16858.143,E2 -16858.143} C_VEL
LIN {X 0,Y 291.41,Z 397.752,A -85,B 0,C 180,E1 -16858.45,E2 -16858.45} C_VEL
LIN {X 0,Y 291.339,Z 397.687,A -85,B 0,C 180,E1 -16862.404,E2 -16862.404} C_VEL
LIN {X 0,Y 291.38,Z 397.658,A -85,B 0,C 180,E1 -16865.37,E2 -16865.37} C_VEL
LIN {X 0,Y 291.375,Z 397.685,A -85,B 0,C 180,E1 -16868.837,E2 -16868.837} C_VEL
LIN {X 0,Y 291.314,Z 397.644,A -85,B 0,C 180,E1 -16872.492,E2 -16872.492} C_VEL
LIN {X 0,Y 291.336,Z 397.695,A -85,B 0,C 180,E1 -16876.359,E2 -16876.359} C_VEL
LIN {X 0,Y 291.392,Z 397.677,A -85,B 0,C 180,E1 -16880.514,E2 -16880.514} C_VEL
LIN {X 0,Y 291.427,Z 397.682,A -85,B 0,C 180,E1 -16882.924,E2 -16882.924} C_VEL
LIN {X 0,Y 291.338,Z 397.676,A -85,B 0,C 180,E1 -16886.302,E2 -16886.302} C_VEL
LIN {X 0,Y 291.381,Z 397.683,A -85,B 0,C 180,E1 -16890.26,E2 -16890.26} C_VEL
LIN {X 0,Y 291.41,Z 397.671,A -85,B 0,C 180,E1 -16894.272,E2 -16894.272} C_VEL
LIN {X 0,Y 291.376,Z 397.687,A -85,B 0,C 180,E1 -16897.3,E2 -16897.3} C_VEL
LIN {X 0,Y 291.452,Z 397.649,A -85,B 0,C 180,E1 -16900.271,E2 -16900.271} C_VEL
LIN {X 0,Y 291.549,Z 397.669,A -85,B 0,C 180,E1 -16904.624,E2 -16904.624} C_VEL
LIN {X 0,Y 291.532,Z 397.638,A -85,B 0,C 180,E1 -16908.881,E2 -16908.881} C_VEL
LIN {X 0,Y 291.704,Z 397.628,A -85,B 0,C 180,E1 -16911.689,E2 -16911.689} C_VEL
LIN {X 0,Y 291.626,Z 397.66,A -85,B 0,C 180,E1 -16914.469,E2 -16914.469} C_VEL
LIN {X 0,Y 291.885,Z 397.591,A -85,B 0,C 180,E1 -16918.621,E2 -16918.621} C_VEL
LIN {X 0,Y 291.885,Z 397.603,A -85,B 0,C 180,E1 -16921.38,E2 -16921.38} C_VEL
LIN {X 0,Y 291.742,Z 397.63,A -85,B 0,C 180,E1 -16926.919,E2 -16926.919} C_VEL
LIN {X 0,Y 291.625,Z 397.618,A -85,B 0,C 180,E1 -16929.713,E2 -16929.713} C_VEL
LIN {X 0,Y 291.513,Z 397.669,A -85,B 0,C 180,E1 -16933.875,E2 -16933.875} C_VEL
LIN {X 0,Y 290.879,Z 397.753,A -85,B 0,C 180,E1 -16935.028,E2 -16935.028} C_VEL
LIN {X 0,Y 287.97,Z 398.098,A -85,B 0,C 180,E1 -16936.902,E2 -16936.902} C_VEL
LIN {X 0,Y 285.491,Z 398.391,A -85,B 0,C 180,E1 -16938.425,E2 -16938.425} C_VEL
LIN {X 0,Y 284.45,Z 398.523,A -85,B 0,C 180,E1 -16939.606,E2 -16939.606} C_VEL
LIN {X 0,Y 284.38,Z 398.535,A -85,B 0,C 180,E1 -16940.007,E2 -16940.007} C_VEL
LIN {X 0,Y 284.366,Z 398.558,A -85,B 0,C 180,E1 -16943.876,E2 -16943.876} C_VEL
LIN {X 0,Y 284.395,Z 398.53,A -85,B 0,C 180,E1 -16947.175,E2 -16947.175} C_VEL
LIN {X 0,Y 284.296,Z 398.57,A -85,B 0,C 180,E1 -16951.275,E2 -16951.275} C_VEL
LIN {X 0,Y 284.361,Z 398.551,A -85,B 0,C 180,E1 -16955.355,E2 -16955.355} C_VEL
LIN {X 0,Y 284.336,Z 398.562,A -85,B 0,C 180,E1 -16958.166,E2 -16958.166} C_VEL
LIN {X 0,Y 284.343,Z 398.568,A -85,B 0,C 180,E1 -16962.142,E2 -16962.142} C_VEL
LIN {X 0,Y 284.297,Z 398.575,A -85,B 0,C 180,E1 -16966.199,E2 -16966.199} C_VEL
LIN {X 0,Y 284.307,Z 398.543,A -85,B 0,C 180,E1 -16970.025,E2 -16970.025} C_VEL
LIN {X 0,Y 284.407,Z 398.784,A -85,B 0,C 180,E1 -16973.516,E2 -16973.516} C_VEL
LIN {X 0,Y 286.131,Z 407.073,A -85,B 0,C 180,E1 -16977.292,E2 -16977.292} C_VEL
LIN {X 0,Y 287.668,Z 414.941,A -85,B 0,C 180,E1 -16980.751,E2 -16980.751} C_VEL
LIN {X 0,Y 288.069,Z 417.213,A -85,B 0,C 180,E1 -16981.592,E2 -16981.592} C_VEL
LIN {X 0,Y 290.683,Z 424.501,A -85,B 0,C 180,E1 -16982.114,E2 -16982.114} C_VEL
LIN {X 0,Y 295.843,Z 449.198,A -85,B 0,C 180,E1 -16983.295,E2 -16983.295} C_VEL
LIN {X 0,Y 298.305,Z 464.606,A -85,B 0,C 180,E1 -16983.935,E2 -16983.935} C_VEL
LIN {X 0,Y 296.616,Z 523.309,A -85,B 0,C 180,E1 -16985.364,E2 -16985.364} C_VEL
LIN {X 0,Y 296.04,Z 532.761,A -85,B 0,C 180,E1 -16985.733,E2 -16985.733} C_VEL
LIN {X 0,Y 295.168,Z 541.882,A -85,B 0,C 180,E1 -16986.217,E2 -16986.217} C_VEL
LIN {X 0,Y 294.033,Z 552.236,A -85,B 0,C 180,E1 -16986.959,E2 -16986.959} C_VEL
LIN {X 0,Y 292.903,Z 561.382,A -85,B 0,C 180,E1 -16987.796,E2 -16987.796} C_VEL
LIN {X 0,Y 291.511,Z 570.38,A -85,B 0,C 180,E1 -16988.8,E2 -16988.8} C_VEL
LIN {X 0,Y 290.027,Z 579.103,A -85,B 0,C 180,E1 -16989.985,E2 -16989.985} C_VEL
LIN {X 0,Y 288.74,Z 586.524,A -85,B 0,C 180,E1 -16991.186,E2 -16991.186} C_VEL
LIN {X 0,Y 287.502,Z 593.96,A -85,B 0,C 180,E1 -16992.623,E2 -16992.623} C_VEL
LIN {X 0,Y 286.142,Z 601.312,A -85,B 0,C 180,E1 -16994.326,E2 -16994.326} C_VEL
LIN {X 0,Y 284.966,Z 607.623,A -85,B 0,C 180,E1 -16996.087,E2 -16996.087} C_VEL
LIN {X 0,Y 283.967,Z 612.896,A -85,B 0,C 180,E1 -16997.857,E2 -16997.857} C_VEL
LIN {X 0,Y 283.179,Z 617.992,A -85,B 0,C 180,E1 -16999.996,E2 -16999.996} C_VEL
